LIN {X 0,Y 154.396,Z 231.863,A -85,B 0,C 180,E1 -25600.747,E2 -25600.747} C_VEL
LIN {X 0,Y 155.915,Z 236.605,A -85,B 0,C 180,E1 -25601.641,E2 -25601.641} C_VEL
LIN {X 0,Y 156.378,Z 245.915,A -85,B 0,C 180,E1 -25602.409,E2 -25602.409} C_VEL
LIN {X 0,Y 153.594,Z 283.863,A -85,B 0,C 180,E1 -25603.923,E2 -25603.923} C_VEL
LIN {X 0,Y 151.68,Z 296.984,A -85,B 0,C 180,E1 -25604.847,E2 -25604.847} C_VEL
LIN {X 0,Y 149.016,Z 309.429,A -85,B 0,C 180,E1 -25606.16,E2 -25606.16} C_VEL
LIN {X 0,Y 145.588,Z 321.476,A -85,B 0,C 180,E1 -25607.953,E2 -25607.953} C_VEL
LIN {X 0,Y 141.539,Z 332.987,A -85,B 0,C 180,E1 -25610.265,E2 -25610.265} C_VEL
LIN {X 0,Y 137.43,Z 343.378,A -85,B 0,C 180,E1 -25613.071,E2 -25613.071} C_VEL
LIN {X 0,Y 133.22,Z 352.693,A -85,B 0,C 180,E1 -25616.367,E2 -25616.367} C_VEL
LIN {X 0,Y 128.946,Z 361.751,A -85,B 0,C 180,E1 -25620.628,E2 -25620.628} C_VEL
LIN {X 0,Y 126.065,Z 367.927,A -85,B 0,C 180,E1 -25624.406,E2 -25624.406} C_VEL
LIN {X 0,Y 122.722,Z 374.878,A -85,B 0,C 180,E1 -25629.907,E2 -25629.907} C_VEL
LIN {X 0,Y 120.764,Z 379.462,A -85,B 0,C 180,E1 -25634.822,E2 -25634.822} C_VEL
LIN {X 0,Y 119.733,Z 382.952,A -85,B 0,C 180,E1 -25639.861,E2 -25639.861} C_VEL
LIN {X 0,Y 119.445,Z 384.69,A -85,B 0,C 180,E1 -25643.245,E2 -25643.245} C_VEL
LIN {X 0,Y 119.517,Z 386.571,A -85,B 0,C 180,E1 -25648.487,E2 -25648.487} C_VEL
LIN {X 0,Y 119.507,Z 387.154,A -85,B 0,C 180,E1 -25651.307,E2 -25651.307} C_VEL
LIN {X 0,Y 119.405,Z 387.457,A -85,B 0,C 180,E1 -25656.763,E2 -25656.763} C_VEL
LIN {X 0,Y 120.43,Z 386.4,A -85,B 0,C 180,E1 -25663.502,E2 -25663.502} C_VEL
LIN {X 0,Y 121.441,Z 385.287,A -85,B 0,C 180,E1 -25666.822,E2 -25666.822} C_VEL
LIN {X 0,Y 122.892,Z 383.731,A -85,B 0,C 180,E1 -25670.071,E2 -25670.071} C_VEL
LIN {X 0,Y 125.89,Z 380.63,A -85,B 0,C 180,E1 -25674.755,E2 -25674.755} C_VEL
LIN {X 0,Y 129.628,Z 376.486,A -85,B 0,C 180,E1 -25679.209,E2 -25679.209} C_VEL
LIN {X 0,Y 132.399,Z 373.117,A -85,B 0,C 180,E1 -25682.022,E2 -25682.022} C_VEL
LIN {X 0,Y 134.104,Z 370.343,A -85,B 0,C 180,E1 -25684.147,E2 -25684.147} C_VEL
LIN {X 0,Y 135.626,Z 365.454,A -85,B 0,C 180,E1 -25687.762,E2 -25687.762} C_VEL
LIN {X 0,Y 137.518,Z 359.972,A -85,B 0,C 180,E1 -25691.126,E2 -25691.126} C_VEL
LIN {X 0,Y 139.702,Z 356.26,A -85,B 0,C 180,E1 -25692.791,E2 -25692.791} C_VEL
LIN {X 0,Y 145.248,Z 347.956,A -85,B 0,C 180,E1 -25695.539,E2 -25695.539} C_VEL
LIN {X 0,Y 151.17,Z 337.757,A -85,B 0,C 180,E1 -25698.063,E2 -25698.063} C_VEL
LIN {X 0,Y 156.791,Z 326.24,A -85,B 0,C 180,E1 -25700.142,E2 -25700.142} C_VEL
LIN {X 0,Y 161.312,Z 314.911,A -85,B 0,C 180,E1 -25701.651,E2 -25701.651} C_VEL
LIN {X 0,Y 164.907,Z 303.329,A -85,B 0,C 180,E1 -25702.792,E2 -25702.792} C_VEL
LIN {X 0,Y 167.865,Z 289.908,A -85,B 0,C 180,E1 -25703.72,E2 -25703.72} C_VEL
LIN {X 0,Y 169.681,Z 276.62,A -85,B 0,C 180,E1 -25704.287,E2 -25704.287} C_VEL
LIN {X 0,Y 171.084,Z 259.051,A -85,B 0,C 180,E1 -25704.893,E2 -25704.893} C_VEL
LIN {X 0,Y 167.769,Z 249.581,A -85,B 0,C 180,E1 -25707.45,E2 -25707.45} C_VEL
LIN {X 0,Y 163.733,Z 239.799,A -85,B 0,C 180,E1 -25710.853,E2 -25710.853} C_VEL
LIN {X 0,Y 160.299,Z 232.342,A -85,B 0,C 180,E1 -25714.165,E2 -25714.165} C_VEL
LIN {X 0,Y 157.633,Z 227.099,A -85,B 0,C 180,E1 -25717.125,E2 -25717.125} C_VEL
LIN {X 0,Y 155.962,Z 224.434,A -85,B 0,C 180,E1 -25719.18,E2 -25719.18} C_VEL
LIN {X 0,Y 153.376,Z 220.422,A -85,B 0,C 180,E1 -25722.984,E2 -25722.984} C_VEL
LIN {X 0,Y 151.058,Z 217.466,A -85,B 0,C 180,E1 -25727.503,E2 -25727.503} C_VEL
LIN {X 0,Y 150.287,Z 215.488,A -85,B 0,C 180,E1 -25729.9,E2 -25729.9} C_VEL
LIN {X 0,Y 149.092,Z 214.312,A -85,B 0,C 180,E1 -25740,E2 -25740} C_VEL
LIN {X 0,Y 150.553,Z 215.702,A -85,B 0,C 180,E1 -25746.534,E2 -25746.534} C_VEL
LIN {X 0,Y 152.095,Z 219.04,A -85,B 0,C 180,E1 -25750.462,E2 -25750.462} C_VEL
LIN {X 0,Y 153.647,Z 220.772,A -85,B 0,C 180,E1 -25753.127,E2 -25753.127} C_VEL
LIN {X 0,Y 156.237,Z 224.739,A -85,B 0,C 180,E1 -25756.833,E2 -25756.833} C_VEL
LIN {X 0,Y 159.48,Z 229.84,A -85,B 0,C 180,E1 -25760.549,E2 -25760.549} C_VEL
LIN {X 0,Y 163.204,Z 235.852,A -85,B 0,C 180,E1 -25764.075,E2 -25764.075} C_VEL
LIN {X 0,Y 167.896,Z 244.453,A -85,B 0,C 180,E1 -25767.873,E2 -25767.873} C_VEL
LIN {X 0,Y 171.689,Z 252.135,A -85,B 0,C 180,E1 -25770.571,E2 -25770.571} C_VEL
LIN {X 0,Y 169.601,Z 275.061,A -85,B 0,C 180,E1 -25771.384,E2 -25771.384} C_VEL
LIN {X 0,Y 167.292,Z 288.542,A -85,B 0,C 180,E1 -25772.211,E2 -25772.211} C_VEL
LIN {X 0,Y 164.053,Z 301.073,A -85,B 0,C 180,E1 -25773.342,E2 -25773.342} C_VEL
LIN {X 0,Y 159.915,Z 313.018,A -85,B 0,C 180,E1 -25774.843,E2 -25774.843} C_VEL
LIN {X 0,Y 154.885,Z 324.813,A -85,B 0,C 180,E1 -25776.891,E2 -25776.891} C_VEL
LIN {X 0,Y 149.638,Z 334.818,A -85,B 0,C 180,E1 -25779.197,E2 -25779.197} C_VEL
LIN {X 0,Y 144.035,Z 343.862,A -85,B 0,C 180,E1 -25781.915,E2 -25781.915} C_VEL
LIN {X 0,Y 138.855,Z 351.308,A -85,B 0,C 180,E1 -25784.877,E2 -25784.877} C_VEL
LIN {X 0,Y 133.231,Z 358.599,A -85,B 0,C 180,E1 -25788.744,E2 -25788.744} C_VEL
LIN {X 0,Y 128.01,Z 364.422,A -85,B 0,C 180,E1 -25792.846,E2 -25792.846} C_VEL
LIN {X 0,Y 123.515,Z 368.987,A -85,B 0,C 180,E1 -25797.276,E2 -25797.276} C_VEL
LIN {X 0,Y 119.689,Z 372.445,A -85,B 0,C 180,E1 -25801.979,E2 -25801.979} C_VEL
LIN {X 0,Y 117.597,Z 374.173,A -85,B 0,C 180,E1 -25805.267,E2 -25805.267} C_VEL
LIN {X 0,Y 114.444,Z 376.385,A -85,B 0,C 180,E1 -25812.115,E2 -25812.115} C_VEL
LIN {X 0,Y 113.499,Z 376.9,A -85,B 0,C 180,E1 -25815.656,E2 -25815.656} C_VEL
LIN {X 0,Y 112.872,Z 376.986,A -85,B 0,C 180,E1 -25819.231,E2 -25819.231} C_VEL
LIN {X 0,Y 112.572,Z 376.683,A -85,B 0,C 180,E1 -25822.824,E2 -25822.824} C_VEL
LIN {X 0,Y 112.532,Z 375.642,A -85,B 0,C 180,E1 -25827.804,E2 -25827.804} C_VEL
LIN {X 0,Y 113.178,Z 373.447,A -85,B 0,C 180,E1 -25833.557,E2 -25833.557} C_VEL
LIN {X 0,Y 114.512,Z 370.428,A -85,B 0,C 180,E1 -25838.823,E2 -25838.823} C_VEL
LIN {X 0,Y 116.535,Z 366.376,A -85,B 0,C 180,E1 -25843.956,E2 -25843.956} C_VEL
LIN {X 0,Y 119.949,Z 360.16,A -85,B 0,C 180,E1 -25849.685,E2 -25849.685} C_VEL
LIN {X 0,Y 123.611,Z 353.4,A -85,B 0,C 180,E1 -25854.34,E2 -25854.34} C_VEL
LIN {X 0,Y 127.95,Z 344.971,A -85,B 0,C 180,E1 -25858.722,E2 -25858.722} C_VEL
LIN {X 0,Y 132.069,Z 336.303,A -85,B 0,C 180,E1 -25862.147,E2 -25862.147} C_VEL
LIN {X 0,Y 136.576,Z 325.633,A -85,B 0,C 180,E1 -25865.37,E2 -25865.37} C_VEL
LIN {X 0,Y 140.367,Z 314.989,A -85,B 0,C 180,E1 -25867.827,E2 -25867.827} C_VEL
LIN {X 0,Y 143.89,Z 303.05,A -85,B 0,C 180,E1 -25869.867,E2 -25869.867} C_VEL
LIN {X 0,Y 146.736,Z 290.607,A -85,B 0,C 180,E1 -25871.415,E2 -25871.415} C_VEL
LIN {X 0,Y 148.853,Z 277.413,A -85,B 0,C 180,E1 -25872.523,E2 -25872.523} C_VEL
LIN {X 0,Y 150.177,Z 262.193,A -85,B 0,C 180,E1 -25873.276,E2 -25873.276} C_VEL
LIN {X 0,Y 152.176,Z 234.348,A -85,B 0,C 180,E1 -25874.363,E2 -25874.363} C_VEL
LIN {X 0,Y 146.942,Z 223.579,A -85,B 0,C 180,E1 -25877.424,E2 -25877.424} C_VEL
LIN {X 0,Y 142.234,Z 215.384,A -85,B 0,C 180,E1 -25880.444,E2 -25880.444} C_VEL
LIN {X 0,Y 137.619,Z 208.218,A -85,B 0,C 180,E1 -25883.771,E2 -25883.771} C_VEL
LIN {X 0,Y 134.714,Z 204.022,A -85,B 0,C 180,E1 -25886.122,E2 -25886.122} C_VEL
LIN {X 0,Y 132.254,Z 200.514,A -85,B 0,C 180,E1 -25888.33,E2 -25888.33} C_VEL
LIN {X 0,Y 129.549,Z 196.833,A -85,B 0,C 180,E1 -25891.04,E2 -25891.04} C_VEL
LIN {X 0,Y 128.745,Z 195.852,A -85,B 0,C 180,E1 -25891.906,E2 -25891.906} C_VEL
LIN {X 0,Y 126.275,Z 193.061,A -85,B 0,C 180,E1 -25894.806,E2 -25894.806} C_VEL
LIN {X 0,Y 125.163,Z 190.919,A -85,B 0,C 180,E1 -25896.417,E2 -25896.417} C_VEL
LIN {X 0,Y 122.32,Z 188.789,A -85,B 0,C 180,E1 -25900.708,E2 -25900.708} C_VEL
LIN {X 0,Y 120.813,Z 185.857,A -85,B 0,C 180,E1 -25904.067,E2 -25904.067} C_VEL
LIN {X 0,Y 120.553,Z 185.187,A -85,B 0,C 180,E1 -25904.791,E2 -25904.791} C_VEL
LIN {X 0,Y 117.979,Z 183.461,A -85,B 0,C 180,E1 -25918.293,E2 -25918.293} C_VEL
LIN {X 0,Y 118.187,Z 183.542,A -85,B 0,C 180,E1 -25920.851,E2 -25920.851} C_VEL
LIN {X 0,Y 120.921,Z 185.41,A -85,B 0,C 180,E1 -25930.436,E2 -25930.436} C_VEL
LIN {X 0,Y 121.931,Z 188.11,A -85,B 0,C 180,E1 -25932.912,E2 -25932.912} C_VEL
LIN {X 0,Y 124.382,Z 190.53,A -85,B 0,C 180,E1 -25936.938,E2 -25936.938} C_VEL
LIN {X 0,Y 125.444,Z 191.294,A -85,B 0,C 180,E1 -25938.369,E2 -25938.369} C_VEL
LIN {X 0,Y 127.207,Z 194.369,A -85,B 0,C 180,E1 -25940.768,E2 -25940.768} C_VEL
LIN {X 0,Y 129.466,Z 196.653,A -85,B 0,C 180,E1 -25943.255,E2 -25943.255} C_VEL
LIN {X 0,Y 132.137,Z 200.357,A -85,B 0,C 180,E1 -25945.952,E2 -25945.952} C_VEL
LIN {X 0,Y 136.383,Z 206.271,A -85,B 0,C 180,E1 -25949.635,E2 -25949.635} C_VEL
LIN {X 0,Y 139.737,Z 211.368,A -85,B 0,C 180,E1 -25952.195,E2 -25952.195} C_VEL
LIN {X 0,Y 143.818,Z 219.923,A -85,B 0,C 180,E1 -25955.15,E2 -25955.15} C_VEL
LIN {X 0,Y 147.828,Z 229.624,A -85,B 0,C 180,E1 -25957.823,E2 -25957.823} C_VEL
LIN {X 0,Y 151.055,Z 238.927,A -85,B 0,C 180,E1 -25959.88,E2 -25959.88} C_VEL
LIN {X 0,Y 151.318,Z 247.608,A -85,B 0,C 180,E1 -25960.581,E2 -25960.581} C_VEL
LIN {X 0,Y 148.549,Z 283.444,A -85,B 0,C 180,E1 -25962.022,E2 -25962.022} C_VEL
LIN {X 0,Y 146.599,Z 296.41,A -85,B 0,C 180,E1 -25962.94,E2 -25962.94} C_VEL
LIN {X 0,Y 143.994,Z 308.361,A -85,B 0,C 180,E1 -25964.209,E2 -25964.209} C_VEL
LIN {X 0,Y 140.384,Z 320.627,A -85,B 0,C 180,E1 -25966.008,E2 -25966.008} C_VEL
LIN {X 0,Y 136.133,Z 332.233,A -85,B 0,C 180,E1 -25968.346,E2 -25968.346} C_VEL
LIN {X 0,Y 131.799,Z 342.7,A -85,B 0,C 180,E1 -25971.208,E2 -25971.208} C_VEL
LIN {X 0,Y 127.328,Z 352.097,A -85,B 0,C 180,E1 -25974.585,E2 -25974.585} C_VEL
LIN {X 0,Y 122.771,Z 361.201,A -85,B 0,C 180,E1 -25978.993,E2 -25978.993} C_VEL
LIN {X 0,Y 119.049,Z 368.542,A -85,B 0,C 180,E1 -25983.724,E2 -25983.724} C_VEL
LIN {X 0,Y 116.032,Z 374.411,A -85,B 0,C 180,E1 -25988.694,E2 -25988.694} C_VEL
LIN {X 0,Y 113.887,Z 379.029,A -85,B 0,C 180,E1 -25993.881,E2 -25993.881} C_VEL
LIN {X 0,Y 112.724,Z 382.546,A -85,B 0,C 180,E1 -25999.223,E2 -25999.223} C_VEL
LIN {X 0,Y 112.361,Z 384.304,A -85,B 0,C 180,E1 -26002.817,E2 -26002.817} C_VEL
LIN {X 0,Y 112.459,Z 386.396,A -85,B 0,C 180,E1 -26009.198,E2 -26009.198} C_VEL
LIN {X 0,Y 112.333,Z 387.077,A -85,B 0,C 180,E1 -26013.59,E2 -26013.59} C_VEL
LIN {X 0,Y 112.722,Z 386.814,A -85,B 0,C 180,E1 -26020.784,E2 -26020.784} C_VEL
LIN {X 0,Y 114.619,Z 385.013,A -85,B 0,C 180,E1 -26027.856,E2 -26027.856} C_VEL
LIN {X 0,Y 116.233,Z 383.48,A -85,B 0,C 180,E1 -26031.275,E2 -26031.275} C_VEL
LIN {X 0,Y 119.435,Z 380.407,A -85,B 0,C 180,E1 -26036.192,E2 -26036.192} C_VEL
LIN {X 0,Y 123.44,Z 376.294,A -85,B 0,C 180,E1 -26040.828,E2 -26040.828} C_VEL
LIN {X 0,Y 128.908,Z 370.011,A -85,B 0,C 180,E1 -26045.883,E2 -26045.883} C_VEL
LIN {X 0,Y 134.522,Z 363.203,A -85,B 0,C 180,E1 -26049.794,E2 -26049.794} C_VEL
LIN {X 0,Y 139.702,Z 356.26,A -85,B 0,C 180,E1 -26052.791,E2 -26052.791} C_VEL
LIN {X 0,Y 141.936,Z 352.367,A -85,B 0,C 180,E1 -26054.355,E2 -26054.355} C_VEL
LIN {X 0,Y 144.244,Z 345.749,A -85,B 0,C 180,E1 -26057.168,E2 -26057.168} C_VEL
LIN {X 0,Y 146.516,Z 338.649,A -85,B 0,C 180,E1 -26059.74,E2 -26059.74} C_VEL
LIN {X 0,Y 148.598,Z 333.995,A -85,B 0,C 180,E1 -26060.895,E2 -26060.895} C_VEL
LIN {X 0,Y 153.67,Z 323.487,A -85,B 0,C 180,E1 -26062.624,E2 -26062.624} C_VEL
LIN {X 0,Y 158.3,Z 311.363,A -85,B 0,C 180,E1 -26064.122,E2 -26064.122} C_VEL
LIN {X 0,Y 162.082,Z 298.685,A -85,B 0,C 180,E1 -26065.202,E2 -26065.202} C_VEL
LIN {X 0,Y 164.705,Z 285.496,A -85,B 0,C 180,E1 -26065.988,E2 -26065.988} C_VEL
LIN {X 0,Y 166.668,Z 267.36,A -85,B 0,C 180,E1 -26066.623,E2 -26066.623} C_VEL
LIN {X 0,Y 167.099,Z 261.511,A -85,B 0,C 180,E1 -26066.855,E2 -26066.855} C_VEL
LIN {X 0,Y 163.705,Z 251.8,A -85,B 0,C 180,E1 -26069.758,E2 -26069.758} C_VEL
LIN {X 0,Y 160.092,Z 242.761,A -85,B 0,C 180,E1 -26073.213,E2 -26073.213} C_VEL
LIN {X 0,Y 157.735,Z 237.548,A -85,B 0,C 180,E1 -26075.755,E2 -26075.755} C_VEL
LIN {X 0,Y 155.773,Z 233.325,A -85,B 0,C 180,E1 -26078.159,E2 -26078.159} C_VEL
LIN {X 0,Y 154.088,Z 230.59,A -85,B 0,C 180,E1 -26080.397,E2 -26080.397} C_VEL
LIN {X 0,Y 151.914,Z 227.078,A -85,B 0,C 180,E1 -26083.885,E2 -26083.885} C_VEL
LIN {X 0,Y 149.793,Z 223.969,A -85,B 0,C 180,E1 -26088.498,E2 -26088.498} C_VEL
LIN {X 0,Y 149.319,Z 222.497,A -85,B 0,C 180,E1 -26090.176,E2 -26090.176} C_VEL
LIN {X 0,Y 148.222,Z 221.381,A -85,B 0,C 180,E1 -26100,E2 -26100} C_VEL
LIN {X 0,Y 149.503,Z 222.698,A -85,B 0,C 180,E1 -26106.072,E2 -26106.072} C_VEL
LIN {X 0,Y 150.944,Z 225.915,A -85,B 0,C 180,E1 -26109.971,E2 -26109.971} C_VEL
LIN {X 0,Y 152.366,Z 227.715,A -85,B 0,C 180,E1 -26112.572,E2 -26112.572} C_VEL
LIN {X 0,Y 155.324,Z 232.491,A -85,B 0,C 180,E1 -26116.935,E2 -26116.935} C_VEL
LIN {X 0,Y 157.845,Z 236.636,A -85,B 0,C 180,E1 -26119.91,E2 -26119.91} C_VEL
LIN {X 0,Y 161.138,Z 242.306,A -85,B 0,C 180,E1 -26123.212,E2 -26123.212} C_VEL
LIN {X 0,Y 165.005,Z 249.718,A -85,B 0,C 180,E1 -26126.565,E2 -26126.565} C_VEL
LIN {X 0,Y 167.661,Z 255.284,A -85,B 0,C 180,E1 -26128.632,E2 -26128.632} C_VEL
LIN {X 0,Y 165.761,Z 275.351,A -85,B 0,C 180,E1 -26129.357,E2 -26129.357} C_VEL
LIN {X 0,Y 163.405,Z 288.528,A -85,B 0,C 180,E1 -26130.136,E2 -26130.136} C_VEL
LIN {X 0,Y 160.245,Z 300.653,A -85,B 0,C 180,E1 -26131.212,E2 -26131.212} C_VEL
LIN {X 0,Y 156.006,Z 312.631,A -85,B 0,C 180,E1 -26132.674,E2 -26132.674} C_VEL
LIN {X 0,Y 150.712,Z 324.669,A -85,B 0,C 180,E1 -26134.723,E2 -26134.723} C_VEL
LIN {X 0,Y 145.225,Z 334.786,A -85,B 0,C 180,E1 -26137.01,E2 -26137.01} C_VEL
LIN {X 0,Y 139.362,Z 343.89,A -85,B 0,C 180,E1 -26139.728,E2 -26139.728} C_VEL
LIN {X 0,Y 133.04,Z 352.479,A -85,B 0,C 180,E1 -26143.202,E2 -26143.202} C_VEL
LIN {X 0,Y 126.978,Z 359.811,A -85,B 0,C 180,E1 -26147.308,E2 -26147.308} C_VEL
LIN {X 0,Y 120.689,Z 366.229,A -85,B 0,C 180,E1 -26152.303,E2 -26152.303} C_VEL
LIN {X 0,Y 116.082,Z 370.446,A -85,B 0,C 180,E1 -26156.979,E2 -26156.979} C_VEL
LIN {X 0,Y 113.404,Z 372.675,A -85,B 0,C 180,E1 -26160.275,E2 -26160.275} C_VEL
LIN {X 0,Y 111.122,Z 374.433,A -85,B 0,C 180,E1 -26163.719,E2 -26163.719} C_VEL
LIN {X 0,Y 107.653,Z 376.674,A -85,B 0,C 180,E1 -26170.945,E2 -26170.945} C_VEL
LIN {X 0,Y 106.57,Z 377.209,A -85,B 0,C 180,E1 -26174.702,E2 -26174.702} C_VEL
LIN {X 0,Y 105.858,Z 377.319,A -85,B 0,C 180,E1 -26178.508,E2 -26178.508} C_VEL
LIN {X 0,Y 105.503,Z 377.03,A -85,B 0,C 180,E1 -26182.34,E2 -26182.34} C_VEL
LIN {X 0,Y 105.466,Z 375.819,A -85,B 0,C 180,E1 -26188.325,E2 -26188.325} C_VEL
LIN {X 0,Y 106.095,Z 373.852,A -85,B 0,C 180,E1 -26193.795,E2 -26193.795} C_VEL
LIN {X 0,Y 107.522,Z 370.864,A -85,B 0,C 180,E1 -26199.401,E2 -26199.401} C_VEL
LIN {X 0,Y 109.681,Z 366.845,A -85,B 0,C 180,E1 -26204.847,E2 -26204.847} C_VEL
LIN {X 0,Y 113.311,Z 360.665,A -85,B 0,C 180,E1 -26210.89,E2 -26210.89} C_VEL
LIN {X 0,Y 117.215,Z 353.945,A -85,B 0,C 180,E1 -26215.762,E2 -26215.762} C_VEL
LIN {X 0,Y 121.806,Z 345.588,A -85,B 0,C 180,E1 -26220.318,E2 -26220.318} C_VEL
LIN {X 0,Y 126.159,Z 336.977,A -85,B 0,C 180,E1 -26223.85,E2 -26223.85} C_VEL
LIN {X 0,Y 130.894,Z 326.378,A -85,B 0,C 180,E1 -26227.155,E2 -26227.155} C_VEL
LIN {X 0,Y 134.866,Z 315.848,A -85,B 0,C 180,E1 -26229.665,E2 -26229.665} C_VEL
LIN {X 0,Y 138.557,Z 304.09,A -85,B 0,C 180,E1 -26231.734,E2 -26231.734} C_VEL
LIN {X 0,Y 141.533,Z 291.87,A -85,B 0,C 180,E1 -26233.3,E2 -26233.3} C_VEL
LIN {X 0,Y 143.847,Z 278.493,A -85,B 0,C 180,E1 -26234.474,E2 -26234.474} C_VEL
LIN {X 0,Y 145.295,Z 263.241,A -85,B 0,C 180,E1 -26235.245,E2 -26235.245} C_VEL
LIN {X 0,Y 147.22,Z 236.744,A -85,B 0,C 180,E1 -26236.32,E2 -26236.32} C_VEL
LIN {X 0,Y 142.32,Z 226.723,A -85,B 0,C 180,E1 -26239.469,E2 -26239.469} C_VEL
LIN {X 0,Y 138.007,Z 219.078,A -85,B 0,C 180,E1 -26242.539,E2 -26242.539} C_VEL
LIN {X 0,Y 134.281,Z 213.216,A -85,B 0,C 180,E1 -26245.499,E2 -26245.499} C_VEL
LIN {X 0,Y 131.743,Z 209.345,A -85,B 0,C 180,E1 -26247.76,E2 -26247.76} C_VEL
LIN {X 0,Y 129.879,Z 206.631,A -85,B 0,C 180,E1 -26249.573,E2 -26249.573} C_VEL
LIN {X 0,Y 126.805,Z 202.306,A -85,B 0,C 180,E1 -26252.946,E2 -26252.946} C_VEL
LIN {X 0,Y 124.438,Z 199.456,A -85,B 0,C 180,E1 -26255.939,E2 -26255.939} C_VEL
LIN {X 0,Y 123.218,Z 197.487,A -85,B 0,C 180,E1 -26257.789,E2 -26257.789} C_VEL
LIN {X 0,Y 120.731,Z 195.214,A -85,B 0,C 180,E1 -26261.985,E2 -26261.985} C_VEL
LIN {X 0,Y 119.358,Z 192.153,A -85,B 0,C 180,E1 -26265.507,E2 -26265.507} C_VEL
LIN {X 0,Y 117.085,Z 190.624,A -85,B 0,C 180,E1 -26276.558,E2 -26276.558} C_VEL
LIN {X 0,Y 117.275,Z 190.529,A -85,B 0,C 180,E1 -26280.429,E2 -26280.429} C_VEL
LIN {X 0,Y 119.573,Z 192.251,A -85,B 0,C 180,E1 -26289.408,E2 -26289.408} C_VEL
LIN {X 0,Y 120.835,Z 195.247,A -85,B 0,C 180,E1 -26292.598,E2 -26292.598} C_VEL
LIN {X 0,Y 123.728,Z 198.002,A -85,B 0,C 180,E1 -26297.35,E2 -26297.35} C_VEL
LIN {X 0,Y 125.768,Z 201.304,A -85,B 0,C 180,E1 -26300.228,E2 -26300.228} C_VEL
LIN {X 0,Y 127.435,Z 203.105,A -85,B 0,C 180,E1 -26302.174,E2 -26302.174} C_VEL
LIN {X 0,Y 130.907,Z 208.098,A -85,B 0,C 180,E1 -26305.835,E2 -26305.835} C_VEL
LIN {X 0,Y 133.994,Z 212.655,A -85,B 0,C 180,E1 -26308.636,E2 -26308.636} C_VEL
LIN {X 0,Y 136.711,Z 216.991,A -85,B 0,C 180,E1 -26310.862,E2 -26310.862} C_VEL
LIN {X 0,Y 140.515,Z 225.459,A -85,B 0,C 180,E1 -26313.849,E2 -26313.849} C_VEL
LIN {X 0,Y 144.6,Z 235.956,A -85,B 0,C 180,E1 -26316.79,E2 -26316.79} C_VEL
LIN {X 0,Y 146.355,Z 241.629,A -85,B 0,C 180,E1 -26318.037,E2 -26318.037} C_VEL
LIN {X 0,Y 146.477,Z 248.428,A -85,B 0,C 180,E1 -26318.59,E2 -26318.59} C_VEL
LIN {X 0,Y 143.653,Z 283.313,A -85,B 0,C 180,E1 -26320.013,E2 -26320.013} C_VEL
LIN {X 0,Y 141.588,Z 296.322,A -85,B 0,C 180,E1 -26320.938,E2 -26320.938} C_VEL
LIN {X 0,Y 138.829,Z 308.413,A -85,B 0,C 180,E1 -26322.242,E2 -26322.242} C_VEL
LIN {X 0,Y 135.362,Z 319.771,A -85,B 0,C 180,E1 -26323.918,E2 -26323.918} C_VEL
LIN {X 0,Y 130.904,Z 331.476,A -85,B 0,C 180,E1 -26326.277,E2 -26326.277} C_VEL
LIN {X 0,Y 126.313,Z 342.016,A -85,B 0,C 180,E1 -26329.178,E2 -26329.178} C_VEL
LIN {X 0,Y 121.585,Z 351.498,A -85,B 0,C 180,E1 -26332.637,E2 -26332.637} C_VEL
LIN {X 0,Y 116.703,Z 360.648,A -85,B 0,C 180,E1 -26337.185,E2 -26337.185} C_VEL
LIN {X 0,Y 112.715,Z 368.033,A -85,B 0,C 180,E1 -26342.123,E2 -26342.123} C_VEL
LIN {X 0,Y 109.407,Z 373.939,A -85,B 0,C 180,E1 -26347.334,E2 -26347.334} C_VEL
LIN {X 0,Y 107.026,Z 378.59,A -85,B 0,C 180,E1 -26352.817,E2 -26352.817} C_VEL
LIN {X 0,Y 105.736,Z 382.137,A -85,B 0,C 180,E1 -26358.502,E2 -26358.502} C_VEL
LIN {X 0,Y 105.291,Z 383.919,A -85,B 0,C 180,E1 -26362.332,E2 -26362.332} C_VEL
LIN {X 0,Y 105.243,Z 385.272,A -85,B 0,C 180,E1 -26366.175,E2 -26366.175} C_VEL
LIN {X 0,Y 105.42,Z 386.22,A -85,B 0,C 180,E1 -26370.004,E2 -26370.004} C_VEL
LIN {X 0,Y 105.239,Z 386.739,A -85,B 0,C 180,E1 -26373.833,E2 -26373.833} C_VEL
LIN {X 0,Y 105.742,Z 386.509,A -85,B 0,C 180,E1 -26381.505,E2 -26381.505} C_VEL
LIN {X 0,Y 107.843,Z 384.736,A -85,B 0,C 180,E1 -26389.02,E2 -26389.02} C_VEL
LIN {X 0,Y 109.636,Z 383.23,A -85,B 0,C 180,E1 -26392.623,E2 -26392.623} C_VEL
LIN {X 0,Y 113.07,Z 380.185,A -85,B 0,C 180,E1 -26397.789,E2 -26397.789} C_VEL
LIN {X 0,Y 117.342,Z 376.101,A -85,B 0,C 180,E1 -26402.621,E2 -26402.621} C_VEL
LIN {X 0,Y 123.207,Z 369.854,A -85,B 0,C 180,E1 -26407.825,E2 -26407.825} C_VEL
LIN {X 0,Y 129.131,Z 363.084,A -85,B 0,C 180,E1 -26411.817,E2 -26411.817} C_VEL
LIN {X 0,Y 135.706,Z 354.701,A -85,B 0,C 180,E1 -26415.408,E2 -26415.408} C_VEL
LIN {X 0,Y 141.54,Z 346.081,A -85,B 0,C 180,E1 -26418.146,E2 -26418.146} C_VEL
LIN {X 0,Y 147.798,Z 335.478,A -85,B 0,C 180,E1 -26420.601,E2 -26420.601} C_VEL
LIN {X 0,Y 148.598,Z 333.995,A -85,B 0,C 180,E1 -26420.895,E2 -26420.895} C_VEL
LIN {X 0,Y 150.631,Z 329.187,A -85,B 0,C 180,E1 -26421.965,E2 -26421.965} C_VEL
LIN {X 0,Y 152.667,Z 321.174,A -85,B 0,C 180,E1 -26424.043,E2 -26424.043} C_VEL
LIN {X 0,Y 154.37,Z 312.79,A -85,B 0,C 180,E1 -26425.907,E2 -26425.907} C_VEL
LIN {X 0,Y 155.798,Z 307.406,A -85,B 0,C 180,E1 -26426.628,E2 -26426.628} C_VEL
LIN {X 0,Y 159.435,Z 293.765,A -85,B 0,C 180,E1 -26427.693,E2 -26427.693} C_VEL
LIN {X 0,Y 161.714,Z 281.24,A -85,B 0,C 180,E1 -26428.293,E2 -26428.293} C_VEL
LIN {X 0,Y 163.3,Z 264.164,A -85,B 0,C 180,E1 -26428.906,E2 -26428.906} C_VEL
LIN {X 0,Y 160.421,Z 255.632,A -85,B 0,C 180,E1 -26431.652,E2 -26431.652} C_VEL
LIN {X 0,Y 157.551,Z 247.953,A -85,B 0,C 180,E1 -26434.71,E2 -26434.71} C_VEL
LIN {X 0,Y 154.769,Z 241.392,A -85,B 0,C 180,E1 -26438.108,E2 -26438.108} C_VEL
LIN {X 0,Y 153.092,Z 237.896,A -85,B 0,C 180,E1 -26440.463,E2 -26440.463} C_VEL
LIN {X 0,Y 150.507,Z 233.754,A -85,B 0,C 180,E1 -26444.772,E2 -26444.772} C_VEL
LIN {X 0,Y 148.533,Z 230.359,A -85,B 0,C 180,E1 -26449.655,E2 -26449.655} C_VEL
LIN {X 0,Y 148.297,Z 229.504,A -85,B 0,C 180,E1 -26450.628,E2 -26450.628} C_VEL
LIN {X 0,Y 147.242,Z 228.554,A -85,B 0,C 180,E1 -26457.264,E2 -26457.264} C_VEL
LIN {X 0,Y 147.412,Z 228.599,A -85,B 0,C 180,E1 -26460.683,E2 -26460.683} C_VEL
LIN {X 0,Y 148.456,Z 229.752,A -85,B 0,C 180,E1 -26465.604,E2 -26465.604} C_VEL
LIN {X 0,Y 150.066,Z 233.174,A -85,B 0,C 180,E1 -26470.03,E2 -26470.03} C_VEL
LIN {X 0,Y 151.054,Z 234.527,A -85,B 0,C 180,E1 -26471.915,E2 -26471.915} C_VEL
LIN {X 0,Y 153.596,Z 238.809,A -85,B 0,C 180,E1 -26475.935,E2 -26475.935} C_VEL
LIN {X 0,Y 156.121,Z 243.251,A -85,B 0,C 180,E1 -26479.134,E2 -26479.134} C_VEL
LIN {X 0,Y 159.479,Z 249.482,A -85,B 0,C 180,E1 -26482.692,E2 -26482.692} C_VEL
LIN {X 0,Y 162.988,Z 256.652,A -85,B 0,C 180,E1 -26485.89,E2 -26485.89} C_VEL
LIN {X 0,Y 163.828,Z 258.556,A -85,B 0,C 180,E1 -26486.605,E2 -26486.605} C_VEL
LIN {X 0,Y 162.024,Z 276.337,A -85,B 0,C 180,E1 -26487.261,E2 -26487.261} C_VEL
LIN {X 0,Y 159.544,Z 289.564,A -85,B 0,C 180,E1 -26488.055,E2 -26488.055} C_VEL
LIN {X 0,Y 155.975,Z 302.264,A -85,B 0,C 180,E1 -26489.187,E2 -26489.187} C_VEL
LIN {X 0,Y 151.416,Z 314.413,A -85,B 0,C 180,E1 -26490.702,E2 -26490.702} C_VEL
LIN {X 0,Y 146.112,Z 325.798,A -85,B 0,C 180,E1 -26492.671,E2 -26492.671} C_VEL
LIN {X 0,Y 141.034,Z 334.751,A -85,B 0,C 180,E1 -26494.689,E2 -26494.689} C_VEL
LIN {X 0,Y 134.905,Z 343.918,A -85,B 0,C 180,E1 -26497.392,E2 -26497.392} C_VEL
LIN {X 0,Y 129.14,Z 351.464,A -85,B 0,C 180,E1 -26500.364,E2 -26500.364} C_VEL
LIN {X 0,Y 122.799,Z 358.843,A -85,B 0,C 180,E1 -26504.321,E2 -26504.321} C_VEL
LIN {X 0,Y 116.907,Z 364.744,A -85,B 0,C 180,E1 -26508.599,E2 -26508.599} C_VEL
LIN {X 0,Y 111.707,Z 369.382,A -85,B 0,C 180,E1 -26513.292,E2 -26513.292} C_VEL
LIN {X 0,Y 107.062,Z 373.03,A -85,B 0,C 180,E1 -26518.582,E2 -26518.582} C_VEL
LIN {X 0,Y 104.739,Z 374.694,A -85,B 0,C 180,E1 -26521.982,E2 -26521.982} C_VEL
LIN {X 0,Y 100.913,Z 376.964,A -85,B 0,C 180,E1 -26529.618,E2 -26529.618} C_VEL
LIN {X 0,Y 99.681,Z 377.514,A -85,B 0,C 180,E1 -26533.616,E2 -26533.616} C_VEL
LIN {X 0,Y 98.876,Z 377.652,A -85,B 0,C 180,E1 -26537.684,E2 -26537.684} C_VEL
LIN {X 0,Y 98.444,Z 377.377,A -85,B 0,C 180,E1 -26541.788,E2 -26541.788} C_VEL
LIN {X 0,Y 98.406,Z 375.954,A -85,B 0,C 180,E1 -26549.076,E2 -26549.076} C_VEL
LIN {X 0,Y 99.017,Z 374.256,A -85,B 0,C 180,E1 -26554.066,E2 -26554.066} C_VEL
LIN {X 0,Y 100.547,Z 371.297,A -85,B 0,C 180,E1 -26560.06,E2 -26560.06} C_VEL
LIN {X 0,Y 102.858,Z 367.311,A -85,B 0,C 180,E1 -26565.857,E2 -26565.857} C_VEL
LIN {X 0,Y 106.734,Z 361.17,A -85,B 0,C 180,E1 -26572.244,E2 -26572.244} C_VEL
LIN {X 0,Y 110.888,Z 354.49,A -85,B 0,C 180,E1 -26577.351,E2 -26577.351} C_VEL
LIN {X 0,Y 115.763,Z 346.199,A -85,B 0,C 180,E1 -26582.083,E2 -26582.083} C_VEL
LIN {X 0,Y 120.353,Z 337.653,A -85,B 0,C 180,E1 -26585.724,E2 -26585.724} C_VEL
LIN {X 0,Y 125.353,Z 327.124,A -85,B 0,C 180,E1 -26589.1,E2 -26589.1} C_VEL
LIN {X 0,Y 129.516,Z 316.687,A -85,B 0,C 180,E1 -26591.657,E2 -26591.657} C_VEL
LIN {X 0,Y 133.38,Z 305.131,A -85,B 0,C 180,E1 -26593.75,E2 -26593.75} C_VEL
LIN {X 0,Y 136.506,Z 293.13,A -85,B 0,C 180,E1 -26595.323,E2 -26595.323} C_VEL
LIN {X 0,Y 138.922,Z 280.138,A -85,B 0,C 180,E1 -26596.51,E2 -26596.51} C_VEL
LIN {X 0,Y 140.348,Z 267.315,A -85,B 0,C 180,E1 -26597.233,E2 -26597.233} C_VEL
LIN {X 0,Y 142.527,Z 239.536,A -85,B 0,C 180,E1 -26598.338,E2 -26598.338} C_VEL
LIN {X 0,Y 138.274,Z 230.675,A -85,B 0,C 180,E1 -26601.355,E2 -26601.355} C_VEL
LIN {X 0,Y 134.301,Z 223.397,A -85,B 0,C 180,E1 -26604.482,E2 -26604.482} C_VEL
LIN {X 0,Y 129.875,Z 216.192,A -85,B 0,C 180,E1 -26608.475,E2 -26608.475} C_VEL
LIN {X 0,Y 127.443,Z 212.585,A -85,B 0,C 180,E1 -26610.994,E2 -26610.994} C_VEL
LIN {X 0,Y 124.925,Z 208.793,A -85,B 0,C 180,E1 -26613.993,E2 -26613.993} C_VEL
LIN {X 0,Y 122.478,Z 205.532,A -85,B 0,C 180,E1 -26617.383,E2 -26617.383} C_VEL
LIN {X 0,Y 121.747,Z 204.266,A -85,B 0,C 180,E1 -26618.592,E2 -26618.592} C_VEL
LIN {X 0,Y 119.328,Z 201.834,A -85,B 0,C 180,E1 -26623.011,E2 -26623.011} C_VEL
LIN {X 0,Y 118.174,Z 199.18,A -85,B 0,C 180,E1 -26626.238,E2 -26626.238} C_VEL
LIN {X 0,Y 116.218,Z 197.68,A -85,B 0,C 180,E1 -26636.533,E2 -26636.533} C_VEL
LIN {X 0,Y 116.444,Z 197.703,A -85,B 0,C 180,E1 -26640.864,E2 -26640.864} C_VEL
LIN {X 0,Y 118.356,Z 199.308,A -85,B 0,C 180,E1 -26648.644,E2 -26648.644} C_VEL
LIN {X 0,Y 119.752,Z 202.344,A -85,B 0,C 180,E1 -26652.283,E2 -26652.283} C_VEL
LIN {X 0,Y 122.121,Z 204.742,A -85,B 0,C 180,E1 -26656.4,E2 -26656.4} C_VEL
LIN {X 0,Y 124.296,Z 208.165,A -85,B 0,C 180,E1 -26659.616,E2 -26659.616} C_VEL
LIN {X 0,Y 125.586,Z 209.738,A -85,B 0,C 180,E1 -26661.223,E2 -26661.223} C_VEL
LIN {X 0,Y 128.597,Z 214.258,A -85,B 0,C 180,E1 -26664.627,E2 -26664.627} C_VEL
LIN {X 0,Y 131.672,Z 219.03,A -85,B 0,C 180,E1 -26667.618,E2 -26667.618} C_VEL
LIN {X 0,Y 133.73,Z 222.545,A -85,B 0,C 180,E1 -26669.442,E2 -26669.442} C_VEL
LIN {X 0,Y 137.463,Z 231.436,A -85,B 0,C 180,E1 -26672.631,E2 -26672.631} C_VEL
LIN {X 0,Y 140.931,Z 241.095,A -85,B 0,C 180,E1 -26675.362,E2 -26675.362} C_VEL
LIN {X 0,Y 141.807,Z 244.117,A -85,B 0,C 180,E1 -26676.052,E2 -26676.052} C_VEL
LIN {X 0,Y 141.806,Z 249.704,A -85,B 0,C 180,E1 -26676.493,E2 -26676.493} C_VEL
LIN {X 0,Y 138.998,Z 282.72,A -85,B 0,C 180,E1 -26677.833,E2 -26677.833} C_VEL
LIN {X 0,Y 136.796,Z 296.115,A -85,B 0,C 180,E1 -26678.786,E2 -26678.786} C_VEL
LIN {X 0,Y 133.841,Z 308.464,A -85,B 0,C 180,E1 -26680.127,E2 -26680.127} C_VEL
LIN {X 0,Y 129.929,Z 320.508,A -85,B 0,C 180,E1 -26681.953,E2 -26681.953} C_VEL
LIN {X 0,Y 125.293,Z 332.018,A -85,B 0,C 180,E1 -26684.347,E2 -26684.347} C_VEL
LIN {X 0,Y 120.475,Z 342.405,A -85,B 0,C 180,E1 -26687.306,E2 -26687.306} C_VEL
LIN {X 0,Y 115.988,Z 350.889,A -85,B 0,C 180,E1 -26690.494,E2 -26690.494} C_VEL
LIN {X 0,Y 110.775,Z 360.096,A -85,B 0,C 180,E1 -26695.185,E2 -26695.185} C_VEL
LIN {X 0,Y 107.751,Z 365.244,A -85,B 0,C 180,E1 -26698.552,E2 -26698.552} C_VEL
LIN {X 0,Y 103.949,Z 371.629,A -85,B 0,C 180,E1 -26703.934,E2 -26703.934} C_VEL
LIN {X 0,Y 100.945,Z 376.7,A -85,B 0,C 180,E1 -26709.632,E2 -26709.632} C_VEL
LIN {X 0,Y 99.107,Z 380.638,A -85,B 0,C 180,E1 -26715.633,E2 -26715.633} C_VEL
LIN {X 0,Y 98.249,Z 383.534,A -85,B 0,C 180,E1 -26721.779,E2 -26721.779} C_VEL
LIN {X 0,Y 98.134,Z 384.9,A -85,B 0,C 180,E1 -26725.897,E2 -26725.897} C_VEL
LIN {X 0,Y 98.314,Z 385.862,A -85,B 0,C 180,E1 -26730.004,E2 -26730.004} C_VEL
LIN {X 0,Y 98.133,Z 386.396,A -85,B 0,C 180,E1 -26734.111,E2 -26734.111} C_VEL
LIN {X 0,Y 98.232,Z 386.503,A -85,B 0,C 180,E1 -26738.23,E2 -26738.23} C_VEL
LIN {X 0,Y 99.712,Z 385.522,A -85,B 0,C 180,E1 -26746.379,E2 -26746.379} C_VEL
LIN {X 0,Y 101.121,Z 384.457,A -85,B 0,C 180,E1 -26750.338,E2 -26750.338} C_VEL
LIN {X 0,Y 103.11,Z 382.98,A -85,B 0,C 180,E1 -26754.143,E2 -26754.143} C_VEL
LIN {X 0,Y 106.812,Z 379.96,A -85,B 0,C 180,E1 -26759.573,E2 -26759.573} C_VEL
LIN {X 0,Y 111.396,Z 375.905,A -85,B 0,C 180,E1 -26764.601,E2 -26764.601} C_VEL
LIN {X 0,Y 117.661,Z 369.698,A -85,B 0,C 180,E1 -26769.953,E2 -26769.953} C_VEL
LIN {X 0,Y 123.907,Z 362.965,A -85,B 0,C 180,E1 -26774.016,E2 -26774.016} C_VEL
LIN {X 0,Y 130.82,Z 354.634,A -85,B 0,C 180,E1 -26777.623,E2 -26777.623} C_VEL
LIN {X 0,Y 136.91,Z 346.083,A -85,B 0,C 180,E1 -26780.357,E2 -26780.357} C_VEL
LIN {X 0,Y 143.41,Z 335.546,A -85,B 0,C 180,E1 -26782.786,E2 -26782.786} C_VEL
LIN {X 0,Y 148.787,Z 325.12,A -85,B 0,C 180,E1 -26784.572,E2 -26784.572} C_VEL
LIN {X 0,Y 153.578,Z 313.669,A -85,B 0,C 180,E1 -26786.044,E2 -26786.044} C_VEL
LIN {X 0,Y 155.798,Z 307.406,A -85,B 0,C 180,E1 -26786.628,E2 -26786.628} C_VEL
LIN {X 0,Y 157.128,Z 301.924,A -85,B 0,C 180,E1 -26787.283,E2 -26787.283} C_VEL
LIN {X 0,Y 158.034,Z 289.365,A -85,B 0,C 180,E1 -26789.419,E2 -26789.419} C_VEL
LIN {X 0,Y 158.355,Z 281.929,A -85,B 0,C 180,E1 -26790.389,E2 -26790.389} C_VEL
LIN {X 0,Y 158.685,Z 278.067,A -85,B 0,C 180,E1 -26790.641,E2 -26790.641} C_VEL
LIN {X 0,Y 159.713,Z 266.896,A -85,B 0,C 180,E1 -26791.05,E2 -26791.05} C_VEL
LIN {X 0,Y 156.979,Z 258.476,A -85,B 0,C 180,E1 -26794.009,E2 -26794.009} C_VEL
LIN {X 0,Y 154.347,Z 251.107,A -85,B 0,C 180,E1 -26797.252,E2 -26797.252} C_VEL
LIN {X 0,Y 152.056,Z 245.548,A -85,B 0,C 180,E1 -26800.525,E2 -26800.525} C_VEL
LIN {X 0,Y 150.647,Z 243.109,A -85,B 0,C 180,E1 -26802.764,E2 -26802.764} C_VEL
LIN {X 0,Y 149.322,Z 240.615,A -85,B 0,C 180,E1 -26805.309,E2 -26805.309} C_VEL
LIN {X 0,Y 147.426,Z 237.059,A -85,B 0,C 180,E1 -26810.435,E2 -26810.435} C_VEL
LIN {X 0,Y 147.111,Z 236.331,A -85,B 0,C 180,E1 -26811.76,E2 -26811.76} C_VEL
LIN {X 0,Y 146.484,Z 235.519,A -85,B 0,C 180,E1 -26820,E2 -26820} C_VEL
LIN {X 0,Y 147.388,Z 236.607,A -85,B 0,C 180,E1 -26824.958,E2 -26824.958} C_VEL
LIN {X 0,Y 148.914,Z 240.045,A -85,B 0,C 180,E1 -26829.508,E2 -26829.508} C_VEL
LIN {X 0,Y 149.721,Z 241.267,A -85,B 0,C 180,E1 -26831.165,E2 -26831.165} C_VEL
LIN {X 0,Y 152.178,Z 245.674,A -85,B 0,C 180,E1 -26835.314,E2 -26835.314} C_VEL
LIN {X 0,Y 154.933,Z 250.726,A -85,B 0,C 180,E1 -26838.943,E2 -26838.943} C_VEL
LIN {X 0,Y 158.272,Z 257.576,A -85,B 0,C 180,E1 -26842.606,E2 -26842.606} C_VEL
LIN {X 0,Y 160.247,Z 261.935,A -85,B 0,C 180,E1 -26844.518,E2 -26844.518} C_VEL
LIN {X 0,Y 158.285,Z 278.882,A -85,B 0,C 180,E1 -26845.144,E2 -26845.144} C_VEL
LIN {X 0,Y 155.722,Z 291.215,A -85,B 0,C 180,E1 -26845.907,E2 -26845.907} C_VEL
LIN {X 0,Y 151.891,Z 303.934,A -85,B 0,C 180,E1 -26847.06,E2 -26847.06} C_VEL
LIN {X 0,Y 147.042,Z 316.131,A -85,B 0,C 180,E1 -26848.596,E2 -26848.596} C_VEL
LIN {X 0,Y 141.709,Z 326.88,A -85,B 0,C 180,E1 -26850.488,E2 -26850.488} C_VEL
LIN {X 0,Y 135.796,Z 336.68,A -85,B 0,C 180,E1 -26852.75,E2 -26852.75} C_VEL
LIN {X 0,Y 129.446,Z 345.576,A -85,B 0,C 180,E1 -26855.469,E2 -26855.469} C_VEL
LIN {X 0,Y 122.693,Z 353.796,A -85,B 0,C 180,E1 -26858.911,E2 -26858.911} C_VEL
LIN {X 0,Y 115.789,Z 361.099,A -85,B 0,C 180,E1 -26863.247,E2 -26863.247} C_VEL
LIN {X 0,Y 109.703,Z 366.587,A -85,B 0,C 180,E1 -26867.723,E2 -26867.723} C_VEL
LIN {X 0,Y 104.355,Z 370.872,A -85,B 0,C 180,E1 -26872.687,E2 -26872.687} C_VEL
LIN {X 0,Y 100.723,Z 373.479,A -85,B 0,C 180,E1 -26876.858,E2 -26876.858} C_VEL
LIN {X 0,Y 96.163,Z 376.3,A -85,B 0,C 180,E1 -26883.987,E2 -26883.987} C_VEL
LIN {X 0,Y 92.843,Z 377.818,A -85,B 0,C 180,E1 -26892.371,E2 -26892.371} C_VEL
LIN {X 0,Y 91.896,Z 377.984,A -85,B 0,C 180,E1 -26896.732,E2 -26896.732} C_VEL
LIN {X 0,Y 91.383,Z 377.725,A -85,B 0,C 180,E1 -26901.148,E2 -26901.148} C_VEL
LIN {X 0,Y 91.368,Z 376.188,A -85,B 0,C 180,E1 -26909.55,E2 -26909.55} C_VEL
LIN {X 0,Y 91.944,Z 374.66,A -85,B 0,C 180,E1 -26914.38,E2 -26914.38} C_VEL
LIN {X 0,Y 93.589,Z 371.726,A -85,B 0,C 180,E1 -26920.816,E2 -26920.816} C_VEL
LIN {X 0,Y 96.074,Z 367.771,A -85,B 0,C 180,E1 -26927.01,E2 -26927.01} C_VEL
LIN {X 0,Y 100.227,Z 361.675,A -85,B 0,C 180,E1 -26933.774,E2 -26933.774} C_VEL
LIN {X 0,Y 104.812,Z 354.802,A -85,B 0,C 180,E1 -26939.293,E2 -26939.293} C_VEL
LIN {X 0,Y 109.843,Z 346.8,A -85,B 0,C 180,E1 -26944.04,E2 -26944.04} C_VEL
LIN {X 0,Y 114.7,Z 338.327,A -85,B 0,C 180,E1 -26947.783,E2 -26947.783} C_VEL
LIN {X 0,Y 119.962,Z 327.87,A -85,B 0,C 180,E1 -26951.225,E2 -26951.225} C_VEL
LIN {X 0,Y 124.337,Z 317.524,A -85,B 0,C 180,E1 -26953.817,E2 -26953.817} C_VEL
LIN {X 0,Y 128.386,Z 306.151,A -85,B 0,C 180,E1 -26955.924,E2 -26955.924} C_VEL
LIN {X 0,Y 131.664,Z 294.389,A -85,B 0,C 180,E1 -26957.496,E2 -26957.496} C_VEL
LIN {X 0,Y 134.353,Z 280.572,A -85,B 0,C 180,E1 -26958.796,E2 -26958.796} C_VEL
LIN {X 0,Y 135.859,Z 267.887,A -85,B 0,C 180,E1 -26959.51,E2 -26959.51} C_VEL
LIN {X 0,Y 137.953,Z 242.285,A -85,B 0,C 180,E1 -26960.534,E2 -26960.534} C_VEL
LIN {X 0,Y 134.662,Z 235.181,A -85,B 0,C 180,E1 -26963.124,E2 -26963.124} C_VEL
LIN {X 0,Y 130.754,Z 227.832,A -85,B 0,C 180,E1 -26966.523,E2 -26966.523} C_VEL
LIN {X 0,Y 127.119,Z 221.69,A -85,B 0,C 180,E1 -26970.159,E2 -26970.159} C_VEL
LIN {X 0,Y 125.011,Z 218.393,A -85,B 0,C 180,E1 -26972.567,E2 -26972.567} C_VEL
LIN {X 0,Y 122.971,Z 215.169,A -85,B 0,C 180,E1 -26975.225,E2 -26975.225} C_VEL
LIN {X 0,Y 120.376,Z 211.196,A -85,B 0,C 180,E1 -26979.272,E2 -26979.272} C_VEL
LIN {X 0,Y 117.763,Z 208.083,A -85,B 0,C 180,E1 -26984.587,E2 -26984.587} C_VEL
LIN {X 0,Y 116.975,Z 206.006,A -85,B 0,C 180,E1 -26987.15,E2 -26987.15} C_VEL
LIN {X 0,Y 115.352,Z 204.736,A -85,B 0,C 180,E1 -26996.507,E2 -26996.507} C_VEL
LIN {X 0,Y 115.573,Z 204.782,A -85,B 0,C 180,E1 -27000.871,E2 -27000.871} C_VEL
LIN {X 0,Y 117.167,Z 206.219,A -85,B 0,C 180,E1 -27007.837,E2 -27007.837} C_VEL
LIN {X 0,Y 118.506,Z 209.208,A -85,B 0,C 180,E1 -27011.6,E2 -27011.6} C_VEL
LIN {X 0,Y 120.521,Z 211.418,A -85,B 0,C 180,E1 -27015.375,E2 -27015.375} C_VEL
LIN {X 0,Y 122.839,Z 215.013,A -85,B 0,C 180,E1 -27018.989,E2 -27018.989} C_VEL
LIN {X 0,Y 124.19,Z 217.076,A -85,B 0,C 180,E1 -27020.794,E2 -27020.794} C_VEL
LIN {X 0,Y 126.512,Z 220.676,A -85,B 0,C 180,E1 -27023.56,E2 -27023.56} C_VEL
LIN {X 0,Y 129.918,Z 226.195,A -85,B 0,C 180,E1 -27027.062,E2 -27027.062} C_VEL
LIN {X 0,Y 132.715,Z 232.729,A -85,B 0,C 180,E1 -27029.758,E2 -27029.758} C_VEL
LIN {X 0,Y 136.098,Z 242.32,A -85,B 0,C 180,E1 -27032.793,E2 -27032.793} C_VEL
LIN {X 0,Y 137.474,Z 247.057,A -85,B 0,C 180,E1 -27033.997,E2 -27033.997} C_VEL
LIN {X 0,Y 137.215,Z 252.275,A -85,B 0,C 180,E1 -27034.299,E2 -27034.299} C_VEL
LIN {X 0,Y 134.49,Z 282.692,A -85,B 0,C 180,E1 -27035.544,E2 -27035.544} C_VEL
LIN {X 0,Y 132.156,Z 296.164,A -85,B 0,C 180,E1 -27036.503,E2 -27036.503} C_VEL
LIN {X 0,Y 129.041,Z 308.499,A -85,B 0,C 180,E1 -27037.847,E2 -27037.847} C_VEL
LIN {X 0,Y 125.271,Z 319.651,A -85,B 0,C 180,E1 -27039.525,E2 -27039.525} C_VEL
LIN {X 0,Y 120.424,Z 331.26,A -85,B 0,C 180,E1 -27041.924,E2 -27041.924} C_VEL
LIN {X 0,Y 115.33,Z 341.722,A -85,B 0,C 180,E1 -27044.9,E2 -27044.9} C_VEL
LIN {X 0,Y 110.584,Z 350.272,A -85,B 0,C 180,E1 -27048.146,E2 -27048.146} C_VEL
LIN {X 0,Y 105.871,Z 358.165,A -85,B 0,C 180,E1 -27052.123,E2 -27052.123} C_VEL
LIN {X 0,Y 101.011,Z 365.874,A -85,B 0,C 180,E1 -27057.374,E2 -27057.374} C_VEL
LIN {X 0,Y 96.389,Z 372.984,A -85,B 0,C 180,E1 -27064.062,E2 -27064.062} C_VEL
LIN {X 0,Y 93.451,Z 377.7,A -85,B 0,C 180,E1 -27070.224,E2 -27070.224} C_VEL
LIN {X 0,Y 91.78,Z 381.307,A -85,B 0,C 180,E1 -27076.723,E2 -27076.723} C_VEL
LIN {X 0,Y 91.205,Z 383.149,A -85,B 0,C 180,E1 -27081.139,E2 -27081.139} C_VEL
LIN {X 0,Y 91.054,Z 384.529,A -85,B 0,C 180,E1 -27085.577,E2 -27085.577} C_VEL
LIN {X 0,Y 91.218,Z 385.505,A -85,B 0,C 180,E1 -27090.004,E2 -27090.004} C_VEL
LIN {X 0,Y 91.052,Z 386.052,A -85,B 0,C 180,E1 -27094.431,E2 -27094.431} C_VEL
LIN {X 0,Y 91.195,Z 386.185,A -85,B 0,C 180,E1 -27098.87,E2 -27098.87} C_VEL
LIN {X 0,Y 92.895,Z 385.23,A -85,B 0,C 180,E1 -27107.619,E2 -27107.619} C_VEL
LIN {X 0,Y 94.462,Z 384.179,A -85,B 0,C 180,E1 -27111.843,E2 -27111.843} C_VEL
LIN {X 0,Y 96.639,Z 382.728,A -85,B 0,C 180,E1 -27115.875,E2 -27115.875} C_VEL
LIN {X 0,Y 100.676,Z 379.731,A -85,B 0,C 180,E1 -27121.575,E2 -27121.575} C_VEL
LIN {X 0,Y 106.509,Z 374.89,A -85,B 0,C 180,E1 -27127.645,E2 -27127.645} C_VEL
LIN {X 0,Y 113.358,Z 368.528,A -85,B 0,C 180,E1 -27133.002,E2 -27133.002} C_VEL
LIN {X 0,Y 120.07,Z 361.61,A -85,B 0,C 180,E1 -27137.029,E2 -27137.029} C_VEL
LIN {X 0,Y 127.366,Z 352.972,A -85,B 0,C 180,E1 -27140.584,E2 -27140.584} C_VEL
LIN {X 0,Y 133.864,Z 344.133,A -85,B 0,C 180,E1 -27143.195,E2 -27143.195} C_VEL
LIN {X 0,Y 140.609,Z 333.268,A -85,B 0,C 180,E1 -27145.563,E2 -27145.563} C_VEL
LIN {X 0,Y 146.233,Z 322.319,A -85,B 0,C 180,E1 -27147.255,E2 -27147.255} C_VEL
LIN {X 0,Y 151.188,Z 310.062,A -85,B 0,C 180,E1 -27148.671,E2 -27148.671} C_VEL
LIN {X 0,Y 154.794,Z 298.489,A -85,B 0,C 180,E1 -27149.618,E2 -27149.618} C_VEL
LIN {X 0,Y 157.665,Z 285.262,A -85,B 0,C 180,E1 -27150.364,E2 -27150.364} C_VEL
LIN {X 0,Y 158.685,Z 278.067,A -85,B 0,C 180,E1 -27150.641,E2 -27150.641} C_VEL
LIN {X 0,Y 158.714,Z 274.991,A -85,B 0,C 180,E1 -27150.971,E2 -27150.971} C_VEL
LIN {X 0,Y 157.956,Z 271.284,A -85,B 0,C 180,E1 -27151.913,E2 -27151.913} C_VEL
LIN {X 0,Y 157.298,Z 269.511,A -85,B 0,C 180,E1 -27152.595,E2 -27152.595} C_VEL
LIN {X 0,Y 154.254,Z 262.877,A -85,B 0,C 180,E1 -27155.865,E2 -27155.865} C_VEL
LIN {X 0,Y 152.054,Z 256.231,A -85,B 0,C 180,E1 -27158.938,E2 -27158.938} C_VEL
LIN {X 0,Y 150.336,Z 251.717,A -85,B 0,C 180,E1 -27161.694,E2 -27161.694} C_VEL
LIN {X 0,Y 148.04,Z 247.349,A -85,B 0,C 180,E1 -27166.088,E2 -27166.088} C_VEL
LIN {X 0,Y 146.25,Z 243.409,A -85,B 0,C 180,E1 -27171.711,E2 -27171.711} C_VEL
LIN {X 0,Y 145.614,Z 242.587,A -85,B 0,C 180,E1 -27180,E2 -27180} C_VEL
LIN {X 0,Y 146.371,Z 243.62,A -85,B 0,C 180,E1 -27184.475,E2 -27184.475} C_VEL
LIN {X 0,Y 147.887,Z 247.06,A -85,B 0,C 180,E1 -27189.23,E2 -27189.23} C_VEL
LIN {X 0,Y 148.567,Z 248.339,A -85,B 0,C 180,E1 -27190.735,E2 -27190.735} C_VEL
LIN {X 0,Y 150.525,Z 252.013,A -85,B 0,C 180,E1 -27194.276,E2 -27194.276} C_VEL
LIN {X 0,Y 153.105,Z 257.078,A -85,B 0,C 180,E1 -27197.964,E2 -27197.964} C_VEL
LIN {X 0,Y 156.469,Z 264.557,A -85,B 0,C 180,E1 -27201.919,E2 -27201.919} C_VEL
LIN {X 0,Y 156.82,Z 265.415,A -85,B 0,C 180,E1 -27202.296,E2 -27202.296} C_VEL
LIN {X 0,Y 154.982,Z 280.061,A -85,B 0,C 180,E1 -27202.869,E2 -27202.869} C_VEL
LIN {X 0,Y 152.131,Z 292.78,A -85,B 0,C 180,E1 -27203.663,E2 -27203.663} C_VEL
LIN {X 0,Y 148.007,Z 305.71,A -85,B 0,C 180,E1 -27204.843,E2 -27204.843} C_VEL
LIN {X 0,Y 143.081,Z 317.367,A -85,B 0,C 180,E1 -27206.315,E2 -27206.315} C_VEL
LIN {X 0,Y 137.526,Z 327.958,A -85,B 0,C 180,E1 -27208.168,E2 -27208.168} C_VEL
LIN {X 0,Y 132.066,Z 336.653,A -85,B 0,C 180,E1 -27210.141,E2 -27210.141} C_VEL
LIN {X 0,Y 125.425,Z 345.607,A -85,B 0,C 180,E1 -27212.802,E2 -27212.802} C_VEL
LIN {X 0,Y 118.124,Z 354.107,A -85,B 0,C 180,E1 -27216.323,E2 -27216.323} C_VEL
LIN {X 0,Y 111.006,Z 361.243,A -85,B 0,C 180,E1 -27220.555,E2 -27220.555} C_VEL
LIN {X 0,Y 104.507,Z 366.767,A -85,B 0,C 180,E1 -27225.076,E2 -27225.076} C_VEL
LIN {X 0,Y 98.753,Z 371.086,A -85,B 0,C 180,E1 -27230.166,E2 -27230.166} C_VEL
LIN {X 0,Y 94.452,Z 373.937,A -85,B 0,C 180,E1 -27234.935,E2 -27234.935} C_VEL
LIN {X 0,Y 89.789,Z 376.575,A -85,B 0,C 180,E1 -27241.985,E2 -27241.985} C_VEL
LIN {X 0,Y 86.064,Z 378.121,A -85,B 0,C 180,E1 -27250.931,E2 -27250.931} C_VEL
LIN {X 0,Y 84.959,Z 378.312,A -85,B 0,C 180,E1 -27255.627,E2 -27255.627} C_VEL
LIN {X 0,Y 84.354,Z 378.071,A -85,B 0,C 180,E1 -27260.404,E2 -27260.404} C_VEL
LIN {X 0,Y 84.13,Z 377.449,A -85,B 0,C 180,E1 -27265.204,E2 -27265.204} C_VEL
LIN {X 0,Y 84.34,Z 376.331,A -85,B 0,C 180,E1 -27270.496,E2 -27270.496} C_VEL
LIN {X 0,Y 84.877,Z 375.059,A -85,B 0,C 180,E1 -27274.745,E2 -27274.745} C_VEL
LIN {X 0,Y 86.652,Z 372.15,A -85,B 0,C 180,E1 -27281.694,E2 -27281.694} C_VEL
LIN {X 0,Y 89.336,Z 368.226,A -85,B 0,C 180,E1 -27288.337,E2 -27288.337} C_VEL
LIN {X 0,Y 93.081,Z 363.169,A -85,B 0,C 180,E1 -27294.532,E2 -27294.532} C_VEL
LIN {X 0,Y 97.668,Z 356.805,A -85,B 0,C 180,E1 -27300.241,E2 -27300.241} C_VEL
LIN {X 0,Y 103.096,Z 348.866,A -85,B 0,C 180,E1 -27305.406,E2 -27305.406} C_VEL
LIN {X 0,Y 108.138,Z 340.774,A -85,B 0,C 180,E1 -27309.316,E2 -27309.316} C_VEL
LIN {X 0,Y 113.597,Z 330.906,A -85,B 0,C 180,E1 -27312.881,E2 -27312.881} C_VEL
LIN {X 0,Y 118.791,Z 319.768,A -85,B 0,C 180,E1 -27315.83,E2 -27315.83} C_VEL
LIN {X 0,Y 122.993,Z 308.865,A -85,B 0,C 180,E1 -27317.968,E2 -27317.968} C_VEL
LIN {X 0,Y 126.676,Z 296.808,A -85,B 0,C 180,E1 -27319.711,E2 -27319.711} C_VEL
LIN {X 0,Y 129.617,Z 283.579,A -85,B 0,C 180,E1 -27321.011,E2 -27321.011} C_VEL
LIN {X 0,Y 131.446,Z 270.071,A -85,B 0,C 180,E1 -27321.855,E2 -27321.855} C_VEL
LIN {X 0,Y 133.543,Z 244.924,A -85,B 0,C 180,E1 -27322.917,E2 -27322.917} C_VEL
LIN {X 0,Y 129.681,Z 236.623,A -85,B 0,C 180,E1 -27326.387,E2 -27326.387} C_VEL
LIN {X 0,Y 126.213,Z 230.187,A -85,B 0,C 180,E1 -27329.923,E2 -27329.923} C_VEL
LIN {X 0,Y 123.192,Z 224.952,A -85,B 0,C 180,E1 -27333.533,E2 -27333.533} C_VEL
LIN {X 0,Y 120.953,Z 221.352,A -85,B 0,C 180,E1 -27336.681,E2 -27336.681} C_VEL
LIN {X 0,Y 118.611,Z 217.555,A -85,B 0,C 180,E1 -27340.742,E2 -27340.742} C_VEL
LIN {X 0,Y 116.501,Z 214.783,A -85,B 0,C 180,E1 -27345.546,E2 -27345.546} C_VEL
LIN {X 0,Y 115.795,Z 212.918,A -85,B 0,C 180,E1 -27348.08,E2 -27348.08} C_VEL
LIN {X 0,Y 114.486,Z 211.784,A -85,B 0,C 180,E1 -27356.48,E2 -27356.48} C_VEL
LIN {X 0,Y 114.67,Z 211.794,A -85,B 0,C 180,E1 -27360.548,E2 -27360.548} C_VEL
LIN {X 0,Y 115.988,Z 213.098,A -85,B 0,C 180,E1 -27366.96,E2 -27366.96} C_VEL
LIN {X 0,Y 117.394,Z 216.196,A -85,B 0,C 180,E1 -27371.164,E2 -27371.164} C_VEL
LIN {X 0,Y 118.981,Z 218.067,A -85,B 0,C 180,E1 -27374.348,E2 -27374.348} C_VEL
LIN {X 0,Y 121.381,Z 221.841,A -85,B 0,C 180,E1 -27378.323,E2 -27378.323} C_VEL
LIN {X 0,Y 124.515,Z 227.136,A -85,B 0,C 180,E1 -27382.504,E2 -27382.504} C_VEL
LIN {X 0,Y 127.594,Z 232.564,A -85,B 0,C 180,E1 -27385.926,E2 -27385.926} C_VEL
LIN {X 0,Y 130.607,Z 240.743,A -85,B 0,C 180,E1 -27389.104,E2 -27389.104} C_VEL
LIN {X 0,Y 133.301,Z 249.437,A -85,B 0,C 180,E1 -27391.742,E2 -27391.742} C_VEL
LIN {X 0,Y 130.227,Z 282.504,A -85,B 0,C 180,E1 -27393.089,E2 -27393.089} C_VEL
LIN {X 0,Y 127.804,Z 295.925,A -85,B 0,C 180,E1 -27394.035,E2 -27394.035} C_VEL
LIN {X 0,Y 124.461,Z 308.516,A -85,B 0,C 180,E1 -27395.394,E2 -27395.394} C_VEL
LIN {X 0,Y 120.231,Z 320.385,A -85,B 0,C 180,E1 -27397.215,E2 -27397.215} C_VEL
LIN {X 0,Y 115.176,Z 331.801,A -85,B 0,C 180,E1 -27399.618,E2 -27399.618} C_VEL
LIN {X 0,Y 109.832,Z 342.099,A -85,B 0,C 180,E1 -27402.625,E2 -27402.625} C_VEL
LIN {X 0,Y 104.301,Z 351.344,A -85,B 0,C 180,E1 -27406.323,E2 -27406.323} C_VEL
LIN {X 0,Y 98.452,Z 360.359,A -85,B 0,C 180,E1 -27411.352,E2 -27411.352} C_VEL
LIN {X 0,Y 94.304,Z 366.493,A -85,B 0,C 180,E1 -27416.023,E2 -27416.023} C_VEL
LIN {X 0,Y 90.025,Z 372.507,A -85,B 0,C 180,E1 -27422.075,E2 -27422.075} C_VEL
LIN {X 0,Y 86.758,Z 377.254,A -85,B 0,C 180,E1 -27428.626,E2 -27428.626} C_VEL
LIN {X 0,Y 84.832,Z 380.891,A -85,B 0,C 180,E1 -27435.614,E2 -27435.614} C_VEL
LIN {X 0,Y 84.17,Z 382.76,A -85,B 0,C 180,E1 -27440.391,E2 -27440.391} C_VEL
LIN {X 0,Y 83.972,Z 384.158,A -85,B 0,C 180,E1 -27445.204,E2 -27445.204} C_VEL
LIN {X 0,Y 84.133,Z 385.148,A -85,B 0,C 180,E1 -27450.004,E2 -27450.004} C_VEL
LIN {X 0,Y 83.971,Z 385.707,A -85,B 0,C 180,E1 -27454.805,E2 -27454.805} C_VEL
LIN {X 0,Y 84.164,Z 385.864,A -85,B 0,C 180,E1 -27459.618,E2 -27459.618} C_VEL
LIN {X 0,Y 86.134,Z 384.939,A -85,B 0,C 180,E1 -27469.053,E2 -27469.053} C_VEL
LIN {X 0,Y 87.878,Z 383.9,A -85,B 0,C 180,E1 -27473.574,E2 -27473.574} C_VEL
LIN {X 0,Y 90.274,Z 382.472,A -85,B 0,C 180,E1 -27477.851,E2 -27477.851} C_VEL
LIN {X 0,Y 94.684,Z 379.498,A -85,B 0,C 180,E1 -27483.832,E2 -27483.832} C_VEL
LIN {X 0,Y 100.392,Z 375.163,A -85,B 0,C 180,E1 -27489.641,E2 -27489.641} C_VEL
LIN {X 0,Y 107.132,Z 369.387,A -85,B 0,C 180,E1 -27494.851,E2 -27494.851} C_VEL
LIN {X 0,Y 114.102,Z 362.73,A -85,B 0,C 180,E1 -27498.988,E2 -27498.988} C_VEL
LIN {X 0,Y 121.687,Z 354.488,A -85,B 0,C 180,E1 -27502.577,E2 -27502.577} C_VEL
LIN {X 0,Y 128.332,Z 346.069,A -85,B 0,C 180,E1 -27505.235,E2 -27505.235} C_VEL
LIN {X 0,Y 135.314,Z 335.69,A -85,B 0,C 180,E1 -27507.569,E2 -27507.569} C_VEL
LIN {X 0,Y 141.8,Z 324.009,A -85,B 0,C 180,E1 -27509.45,E2 -27509.45} C_VEL
LIN {X 0,Y 146.859,Z 312.4,A -85,B 0,C 180,E1 -27510.855,E2 -27510.855} C_VEL
LIN {X 0,Y 150.615,Z 301.637,A -85,B 0,C 180,E1 -27511.736,E2 -27511.736} C_VEL
LIN {X 0,Y 153.837,Z 288.668,A -85,B 0,C 180,E1 -27512.53,E2 -27512.53} C_VEL
LIN {X 0,Y 155.866,Z 275.539,A -85,B 0,C 180,E1 -27513.039,E2 -27513.039} C_VEL
LIN {X 0,Y 156.349,Z 269.741,A -85,B 0,C 180,E1 -27513.288,E2 -27513.288} C_VEL
LIN {X 0,Y 154.254,Z 262.877,A -85,B 0,C 180,E1 -27515.865,E2 -27515.865} C_VEL
LIN {X 0,Y 152.79,Z 259.8,A -85,B 0,C 180,E1 -27517.67,E2 -27517.67} C_VEL
LIN {X 0,Y 151.179,Z 257.791,A -85,B 0,C 180,E1 -27519.697,E2 -27519.697} C_VEL
LIN {X 0,Y 146.663,Z 253.887,A -85,B 0,C 180,E1 -27527.182,E2 -27527.182} C_VEL
LIN {X 0,Y 145.226,Z 250.355,A -85,B 0,C 180,E1 -27532.353,E2 -27532.353} C_VEL
LIN {X 0,Y 144.746,Z 249.651,A -85,B 0,C 180,E1 -27540,E2 -27540} C_VEL
LIN {X 0,Y 145.402,Z 250.712,A -85,B 0,C 180,E1 -27544.158,E2 -27544.158} C_VEL
LIN {X 0,Y 146.865,Z 254.068,A -85,B 0,C 180,E1 -27548.948,E2 -27548.948} C_VEL
LIN {X 0,Y 149.062,Z 258.672,A -85,B 0,C 180,E1 -27553.462,E2 -27553.462} C_VEL
LIN {X 0,Y 151.263,Z 263.352,A -85,B 0,C 180,E1 -27556.882,E2 -27556.882} C_VEL
LIN {X 0,Y 153.655,Z 268.974,A -85,B 0,C 180,E1 -27560.002,E2 -27560.002} C_VEL
LIN {X 0,Y 151.664,Z 282.437,A -85,B 0,C 180,E1 -27560.564,E2 -27560.564} C_VEL
LIN {X 0,Y 148.47,Z 295.458,A -85,B 0,C 180,E1 -27561.4,E2 -27561.4} C_VEL
LIN {X 0,Y 144.491,Z 307.063,A -85,B 0,C 180,E1 -27562.454,E2 -27562.454} C_VEL
LIN {X 0,Y 139.462,Z 318.344,A -85,B 0,C 180,E1 -27563.866,E2 -27563.866} C_VEL
LIN {X 0,Y 133.58,Z 329.035,A -85,B 0,C 180,E1 -27565.707,E2 -27565.707} C_VEL
LIN {X 0,Y 127.234,Z 338.58,A -85,B 0,C 180,E1 -27567.893,E2 -27567.893} C_VEL
LIN {X 0,Y 120.347,Z 347.266,A -85,B 0,C 180,E1 -27570.525,E2 -27570.525} C_VEL
LIN {X 0,Y 113.564,Z 354.673,A -85,B 0,C 180,E1 -27573.653,E2 -27573.653} C_VEL
LIN {X 0,Y 106.477,Z 361.388,A -85,B 0,C 180,E1 -27577.617,E2 -27577.617} C_VEL
LIN {X 0,Y 99.567,Z 366.947,A -85,B 0,C 180,E1 -27582.166,E2 -27582.166} C_VEL
LIN {X 0,Y 93.356,Z 371.3,A -85,B 0,C 180,E1 -27587.344,E2 -27587.344} C_VEL
LIN {X 0,Y 88.248,Z 374.409,A -85,B 0,C 180,E1 -27592.789,E2 -27592.789} C_VEL
LIN {X 0,Y 83.546,Z 376.85,A -85,B 0,C 180,E1 -27599.682,E2 -27599.682} C_VEL
LIN {X 0,Y 79.335,Z 378.426,A -85,B 0,C 180,E1 -27609.242,E2 -27609.242} C_VEL
LIN {X 0,Y 78.072,Z 378.635,A -85,B 0,C 180,E1 -27614.328,E2 -27614.328} C_VEL
LIN {X 0,Y 77.332,Z 378.418,A -85,B 0,C 180,E1 -27619.523,E2 -27619.523} C_VEL
LIN {X 0,Y 77.054,Z 377.809,A -85,B 0,C 180,E1 -27624.762,E2 -27624.762} C_VEL
LIN {X 0,Y 77.333,Z 376.503,A -85,B 0,C 180,E1 -27631.426,E2 -27631.426} C_VEL
LIN {X 0,Y 78.944,Z 373.629,A -85,B 0,C 180,E1 -27640.251,E2 -27640.251} C_VEL
LIN {X 0,Y 81.574,Z 370.088,A -85,B 0,C 180,E1 -27647.545,E2 -27647.545} C_VEL
LIN {X 0,Y 85.2,Z 365.456,A -85,B 0,C 180,E1 -27654.353,E2 -27654.353} C_VEL
LIN {X 0,Y 90.738,Z 358.478,A -85,B 0,C 180,E1 -27661.516,E2 -27661.516} C_VEL
LIN {X 0,Y 96.41,Z 350.919,A -85,B 0,C 180,E1 -27666.965,E2 -27666.965} C_VEL
LIN {X 0,Y 102.775,Z 341.415,A -85,B 0,C 180,E1 -27671.81,E2 -27671.81} C_VEL
LIN {X 0,Y 108.525,Z 331.611,A -85,B 0,C 180,E1 -27675.421,E2 -27675.421} C_VEL
LIN {X 0,Y 113.996,Z 320.599,A -85,B 0,C 180,E1 -27678.37,E2 -27678.37} C_VEL
LIN {X 0,Y 118.396,Z 309.817,A -85,B 0,C 180,E1 -27680.499,E2 -27680.499} C_VEL
LIN {X 0,Y 122.251,Z 297.934,A -85,B 0,C 180,E1 -27682.223,E2 -27682.223} C_VEL
LIN {X 0,Y 125.274,Z 285.309,A -85,B 0,C 180,E1 -27683.514,E2 -27683.514} C_VEL
LIN {X 0,Y 127.298,Z 271.843,A -85,B 0,C 180,E1 -27684.38,E2 -27684.38} C_VEL
LIN {X 0,Y 129.471,Z 247.868,A -85,B 0,C 180,E1 -27685.361,E2 -27685.361} C_VEL
LIN {X 0,Y 126.036,Z 240.323,A -85,B 0,C 180,E1 -27688.86,E2 -27688.86} C_VEL
LIN {X 0,Y 122.377,Z 233.332,A -85,B 0,C 180,E1 -27693.204,E2 -27693.204} C_VEL
LIN {X 0,Y 119.418,Z 228.05,A -85,B 0,C 180,E1 -27697.54,E2 -27697.54} C_VEL
LIN {X 0,Y 117.111,Z 224.2,A -85,B 0,C 180,E1 -27701.855,E2 -27701.855} C_VEL
LIN {X 0,Y 115.14,Z 221.154,A -85,B 0,C 180,E1 -27706.993,E2 -27706.993} C_VEL
LIN {X 0,Y 114.696,Z 219.849,A -85,B 0,C 180,E1 -27708.85,E2 -27708.85} C_VEL
LIN {X 0,Y 113.62,Z 218.84,A -85,B 0,C 180,E1 -27716.453,E2 -27716.453} C_VEL
LIN {X 0,Y 113.86,Z 218.946,A -85,B 0,C 180,E1 -27721.105,E2 -27721.105} C_VEL
LIN {X 0,Y 114.858,Z 220.008,A -85,B 0,C 180,E1 -27726.147,E2 -27726.147} C_VEL
LIN {X 0,Y 116.401,Z 223.334,A -85,B 0,C 180,E1 -27730.986,E2 -27730.986} C_VEL
LIN {X 0,Y 117.574,Z 224.949,A -85,B 0,C 180,E1 -27733.503,E2 -27733.503} C_VEL
LIN {X 0,Y 120.119,Z 229.27,A -85,B 0,C 180,E1 -27737.971,E2 -27737.971} C_VEL
LIN {X 0,Y 123.272,Z 234.782,A -85,B 0,C 180,E1 -27742.302,E2 -27742.302} C_VEL
LIN {X 0,Y 125.161,Z 238.777,A -85,B 0,C 180,E1 -27744.588,E2 -27744.588} C_VEL
LIN {X 0,Y 127.941,Z 247.236,A -85,B 0,C 180,E1 -27747.836,E2 -27747.836} C_VEL
LIN {X 0,Y 129.198,Z 251.632,A -85,B 0,C 180,E1 -27749.222,E2 -27749.222} C_VEL
LIN {X 0,Y 126.313,Z 281.772,A -85,B 0,C 180,E1 -27750.452,E2 -27750.452} C_VEL
LIN {X 0,Y 123.857,Z 294.976,A -85,B 0,C 180,E1 -27751.335,E2 -27751.335} C_VEL
LIN {X 0,Y 120.485,Z 307.469,A -85,B 0,C 180,E1 -27752.639,E2 -27752.639} C_VEL
LIN {X 0,Y 116.054,Z 319.521,A -85,B 0,C 180,E1 -27754.408,E2 -27754.408} C_VEL
LIN {X 0,Y 110.763,Z 331.036,A -85,B 0,C 180,E1 -27756.774,E2 -27756.774} C_VEL
LIN {X 0,Y 105.151,Z 341.426,A -85,B 0,C 180,E1 -27759.776,E2 -27759.776} C_VEL
LIN {X 0,Y 99.27,Z 350.743,A -85,B 0,C 180,E1 -27763.482,E2 -27763.482} C_VEL
LIN {X 0,Y 92.875,Z 359.937,A -85,B 0,C 180,E1 -27768.688,E2 -27768.688} C_VEL
LIN {X 0,Y 88.403,Z 365.982,A -85,B 0,C 180,E1 -27773.417,E2 -27773.417} C_VEL
LIN {X 0,Y 83.766,Z 372.027,A -85,B 0,C 180,E1 -27779.78,E2 -27779.78} C_VEL
LIN {X 0,Y 80.154,Z 376.809,A -85,B 0,C 180,E1 -27786.766,E2 -27786.766} C_VEL
LIN {X 0,Y 77.935,Z 380.476,A -85,B 0,C 180,E1 -27794.309,E2 -27794.309} C_VEL
LIN {X 0,Y 77.137,Z 382.368,A -85,B 0,C 180,E1 -27799.506,E2 -27799.506} C_VEL
LIN {X 0,Y 76.886,Z 383.787,A -85,B 0,C 180,E1 -27804.76,E2 -27804.76} C_VEL
LIN {X 0,Y 77.05,Z 384.792,A -85,B 0,C 180,E1 -27810.005,E2 -27810.005} C_VEL
LIN {X 0,Y 76.885,Z 385.363,A -85,B 0,C 180,E1 -27815.249,E2 -27815.249} C_VEL
LIN {X 0,Y 77.166,Z 385.54,A -85,B 0,C 180,E1 -27820.5,E2 -27820.5} C_VEL
LIN {X 0,Y 79.423,Z 384.647,A -85,B 0,C 180,E1 -27830.734,E2 -27830.734} C_VEL
LIN {X 0,Y 81.391,Z 383.623,A -85,B 0,C 180,E1 -27835.583,E2 -27835.583} C_VEL
LIN {X 0,Y 84.035,Z 382.213,A -85,B 0,C 180,E1 -27840.123,E2 -27840.123} C_VEL
LIN {X 0,Y 88.861,Z 379.264,A -85,B 0,C 180,E1 -27846.387,E2 -27846.387} C_VEL
LIN {X 0,Y 94.555,Z 375.295,A -85,B 0,C 180,E1 -27851.99,E2 -27851.99} C_VEL
LIN {X 0,Y 101.033,Z 370.209,A -85,B 0,C 180,E1 -27856.924,E2 -27856.924} C_VEL
LIN {X 0,Y 108.303,Z 363.847,A -85,B 0,C 180,E1 -27861.146,E2 -27861.146} C_VEL
LIN {X 0,Y 116.175,Z 355.905,A -85,B 0,C 180,E1 -27864.758,E2 -27864.758} C_VEL
LIN {X 0,Y 123.009,Z 347.832,A -85,B 0,C 180,E1 -27867.434,E2 -27867.434} C_VEL
LIN {X 0,Y 130.18,Z 338.001,A -85,B 0,C 180,E1 -27869.749,E2 -27869.749} C_VEL
LIN {X 0,Y 136.826,Z 327.018,A -85,B 0,C 180,E1 -27871.601,E2 -27871.601} C_VEL
LIN {X 0,Y 142.084,Z 316.264,A -85,B 0,C 180,E1 -27872.921,E2 -27872.921} C_VEL
LIN {X 0,Y 146.238,Z 305.68,A -85,B 0,C 180,E1 -27873.874,E2 -27873.874} C_VEL
LIN {X 0,Y 150.057,Z 292.454,A -85,B 0,C 180,E1 -27874.772,E2 -27874.772} C_VEL
LIN {X 0,Y 152.444,Z 280.098,A -85,B 0,C 180,E1 -27875.305,E2 -27875.305} C_VEL
LIN {X 0,Y 153.262,Z 272.806,A -85,B 0,C 180,E1 -27875.567,E2 -27875.567} C_VEL
LIN {X 0,Y 150.872,Z 264.445,A -85,B 0,C 180,E1 -27879.067,E2 -27879.067} C_VEL
LIN {X 0,Y 148.863,Z 258.318,A -85,B 0,C 180,E1 -27882.551,E2 -27882.551} C_VEL
LIN {X 0,Y 146.946,Z 254.276,A -85,B 0,C 180,E1 -27886.517,E2 -27886.517} C_VEL
LIN {X 0,Y 146.663,Z 253.887,A -85,B 0,C 180,E1 -27887.182,E2 -27887.182} C_VEL
LIN {X 0,Y 145.775,Z 253.188,A -85,B 0,C 180,E1 -27889.453,E2 -27889.453} C_VEL
LIN {X 0,Y 144.968,Z 253.653,A -85,B 0,C 180,E1 -27891.772,E2 -27891.772} C_VEL
LIN {X 0,Y 143.801,Z 256.511,A -85,B 0,C 180,E1 -27898.062,E2 -27898.062} C_VEL
LIN {X 0,Y 143.847,Z 256.724,A -85,B 0,C 180,E1 -27899.668,E2 -27899.668} C_VEL
LIN {X 0,Y 144.403,Z 257.626,A -85,B 0,C 180,E1 -27903.624,E2 -27903.624} C_VEL
LIN {X 0,Y 146.02,Z 261.73,A -85,B 0,C 180,E1 -27909.174,E2 -27909.174} C_VEL
LIN {X 0,Y 147.857,Z 265.805,A -85,B 0,C 180,E1 -27913.049,E2 -27913.049} C_VEL
LIN {X 0,Y 150.158,Z 271.334,A -85,B 0,C 180,E1 -27916.847,E2 -27916.847} C_VEL
LIN {X 0,Y 150.639,Z 272.708,A -85,B 0,C 180,E1 -27917.599,E2 -27917.599} C_VEL
LIN {X 0,Y 148.328,Z 286.138,A -85,B 0,C 180,E1 -27918.237,E2 -27918.237} C_VEL
LIN {X 0,Y 144.982,Z 298.168,A -85,B 0,C 180,E1 -27919.028,E2 -27919.028} C_VEL
LIN {X 0,Y 140.393,Z 310.326,A -85,B 0,C 180,E1 -27920.177,E2 -27920.177} C_VEL
LIN {X 0,Y 135.114,Z 321.262,A -85,B 0,C 180,E1 -27921.595,E2 -27921.595} C_VEL
LIN {X 0,Y 129.145,Z 331.287,A -85,B 0,C 180,E1 -27923.312,E2 -27923.312} C_VEL
LIN {X 0,Y 122.592,Z 340.469,A -85,B 0,C 180,E1 -27925.45,E2 -27925.45} C_VEL
LIN {X 0,Y 115.478,Z 348.838,A -85,B 0,C 180,E1 -27928.053,E2 -27928.053} C_VEL
LIN {X 0,Y 107.35,Z 356.997,A -85,B 0,C 180,E1 -27931.665,E2 -27931.665} C_VEL
LIN {X 0,Y 99.761,Z 363.539,A -85,B 0,C 180,E1 -27935.884,E2 -27935.884} C_VEL
LIN {X 0,Y 92.601,Z 368.731,A -85,B 0,C 180,E1 -27940.622,E2 -27940.622} C_VEL
LIN {X 0,Y 86.18,Z 372.745,A -85,B 0,C 180,E1 -27946.112,E2 -27946.112} C_VEL
LIN {X 0,Y 80.59,Z 375.698,A -85,B 0,C 180,E1 -27952.373,E2 -27952.373} C_VEL
LIN {X 0,Y 77.448,Z 377.126,A -85,B 0,C 180,E1 -27957.007,E2 -27957.007} C_VEL
LIN {X 0,Y 72.676,Z 378.731,A -85,B 0,C 180,E1 -27967.239,E2 -27967.239} C_VEL
LIN {X 0,Y 71.21,Z 378.955,A -85,B 0,C 180,E1 -27972.772,E2 -27972.772} C_VEL
LIN {X 0,Y 70.329,Z 378.765,A -85,B 0,C 180,E1 -27978.466,E2 -27978.466} C_VEL
LIN {X 0,Y 69.979,Z 378.169,A -85,B 0,C 180,E1 -27984.231,E2 -27984.231} C_VEL
LIN {X 0,Y 70.369,Z 376.567,A -85,B 0,C 180,E1 -27992.86,E2 -27992.86} C_VEL
LIN {X 0,Y 72.837,Z 372.987,A -85,B 0,C 180,E1 -28003.953,E2 -28003.953} C_VEL
LIN {X 0,Y 76.046,Z 369.125,A -85,B 0,C 180,E1 -28011.69,E2 -28011.69} C_VEL
LIN {X 0,Y 80.401,Z 364.143,A -85,B 0,C 180,E1 -28018.73,E2 -28018.73} C_VEL
LIN {X 0,Y 85.754,Z 357.883,A -85,B 0,C 180,E1 -28025.002,E2 -28025.002} C_VEL
LIN {X 0,Y 91.956,Z 350.041,A -85,B 0,C 180,E1 -28030.508,E2 -28030.508} C_VEL
LIN {X 0,Y 97.632,Z 342.055,A -85,B 0,C 180,E1 -28034.569,E2 -28034.569} C_VEL
LIN {X 0,Y 103.688,Z 332.316,A -85,B 0,C 180,E1 -28038.203,E2 -28038.203} C_VEL
LIN {X 0,Y 109.427,Z 321.432,A -85,B 0,C 180,E1 -28041.138,E2 -28041.138} C_VEL
LIN {X 0,Y 114.048,Z 310.769,A -85,B 0,C 180,E1 -28043.229,E2 -28043.229} C_VEL
LIN {X 0,Y 118.404,Z 297.942,A -85,B 0,C 180,E1 -28045.063,E2 -28045.063} C_VEL
LIN {X 0,Y 121.603,Z 284.908,A -85,B 0,C 180,E1 -28046.341,E2 -28046.341} C_VEL
LIN {X 0,Y 123.67,Z 271.373,A -85,B 0,C 180,E1 -28047.166,E2 -28047.166} C_VEL
LIN {X 0,Y 125.551,Z 250.919,A -85,B 0,C 180,E1 -28048.028,E2 -28048.028} C_VEL
LIN {X 0,Y 122.581,Z 244.091,A -85,B 0,C 180,E1 -28051.522,E2 -28051.522} C_VEL
LIN {X 0,Y 119.39,Z 237.638,A -85,B 0,C 180,E1 -28055.954,E2 -28055.954} C_VEL
LIN {X 0,Y 117.437,Z 234.099,A -85,B 0,C 180,E1 -28059.242,E2 -28059.242} C_VEL
LIN {X 0,Y 115.68,Z 230.857,A -85,B 0,C 180,E1 -28062.946,E2 -28062.946} C_VEL
LIN {X 0,Y 113.882,Z 227.612,A -85,B 0,C 180,E1 -28068.348,E2 -28068.348} C_VEL
LIN {X 0,Y 113.697,Z 226.843,A -85,B 0,C 180,E1 -28069.313,E2 -28069.313} C_VEL
LIN {X 0,Y 112.754,Z 225.889,A -85,B 0,C 180,E1 -28076.426,E2 -28076.426} C_VEL
LIN {X 0,Y 112.99,Z 226.016,A -85,B 0,C 180,E1 -28081.113,E2 -28081.113} C_VEL
LIN {X 0,Y 113.784,Z 227.04,A -85,B 0,C 180,E1 -28085.482,E2 -28085.482} C_VEL
LIN {X 0,Y 115.517,Z 230.648,A -85,B 0,C 180,E1 -28091.071,E2 -28091.071} C_VEL
LIN {X 0,Y 116.209,Z 231.832,A -85,B 0,C 180,E1 -28092.664,E2 -28092.664} C_VEL
LIN {X 0,Y 118.329,Z 235.655,A -85,B 0,C 180,E1 -28096.719,E2 -28096.719} C_VEL
LIN {X 0,Y 121.113,Z 240.962,A -85,B 0,C 180,E1 -28100.93,E2 -28100.93} C_VEL
LIN {X 0,Y 122.497,Z 244.076,A -85,B 0,C 180,E1 -28102.784,E2 -28102.784} C_VEL
LIN {X 0,Y 124.949,Z 252.372,A -85,B 0,C 180,E1 -28106.033,E2 -28106.033} C_VEL
LIN {X 0,Y 125.349,Z 253.965,A -85,B 0,C 180,E1 -28106.549,E2 -28106.549} C_VEL
LIN {X 0,Y 122.498,Z 282.098,A -85,B 0,C 180,E1 -28107.694,E2 -28107.694} C_VEL
LIN {X 0,Y 119.989,Z 294.933,A -85,B 0,C 180,E1 -28108.537,E2 -28108.537} C_VEL
LIN {X 0,Y 116.435,Z 307.496,A -85,B 0,C 180,E1 -28109.818,E2 -28109.818} C_VEL
LIN {X 0,Y 112.172,Z 318.656,A -85,B 0,C 180,E1 -28111.396,E2 -28111.396} C_VEL
LIN {X 0,Y 106.636,Z 330.269,A -85,B 0,C 180,E1 -28113.695,E2 -28113.695} C_VEL
LIN {X 0,Y 100.76,Z 340.742,A -85,B 0,C 180,E1 -28116.674,E2 -28116.674} C_VEL
LIN {X 0,Y 94.506,Z 350.141,A -85,B 0,C 180,E1 -28120.344,E2 -28120.344} C_VEL
LIN {X 0,Y 87.748,Z 359.245,A -85,B 0,C 180,E1 -28125.515,E2 -28125.515} C_VEL
LIN {X 0,Y 82.683,Z 365.53,A -85,B 0,C 180,E1 -28130.509,E2 -28130.509} C_VEL
LIN {X 0,Y 77.653,Z 371.545,A -85,B 0,C 180,E1 -28137.116,E2 -28137.116} C_VEL
LIN {X 0,Y 73.657,Z 376.363,A -85,B 0,C 180,E1 -28144.579,E2 -28144.579} C_VEL
LIN {X 0,Y 71.097,Z 380.06,A -85,B 0,C 180,E1 -28152.755,E2 -28152.755} C_VEL
LIN {X 0,Y 70.143,Z 381.971,A -85,B 0,C 180,E1 -28158.446,E2 -28158.446} C_VEL
LIN {X 0,Y 69.794,Z 383.414,A -85,B 0,C 180,E1 -28164.226,E2 -28164.226} C_VEL
LIN {X 0,Y 69.954,Z 384.434,A -85,B 0,C 180,E1 -28170.005,E2 -28170.005} C_VEL
LIN {X 0,Y 69.796,Z 385.017,A -85,B 0,C 180,E1 -28175.784,E2 -28175.784} C_VEL
LIN {X 0,Y 70.172,Z 385.212,A -85,B 0,C 180,E1 -28181.56,E2 -28181.56} C_VEL
LIN {X 0,Y 71.166,Z 384.984,A -85,B 0,C 180,E1 -28187.239,E2 -28187.239} C_VEL
LIN {X 0,Y 75.026,Z 383.345,A -85,B 0,C 180,E1 -28197.934,E2 -28197.934} C_VEL
LIN {X 0,Y 77.954,Z 381.951,A -85,B 0,C 180,E1 -28202.752,E2 -28202.752} C_VEL
LIN {X 0,Y 83.236,Z 379.029,A -85,B 0,C 180,E1 -28209.296,E2 -28209.296} C_VEL
LIN {X 0,Y 89.377,Z 375.09,A -85,B 0,C 180,E1 -28215.053,E2 -28215.053} C_VEL
LIN {X 0,Y 96.312,Z 370.038,A -85,B 0,C 180,E1 -28220.019,E2 -28220.019} C_VEL
LIN {X 0,Y 103.997,Z 363.721,A -85,B 0,C 180,E1 -28224.193,E2 -28224.193} C_VEL
LIN {X 0,Y 112.214,Z 355.832,A -85,B 0,C 180,E1 -28227.731,E2 -28227.731} C_VEL
LIN {X 0,Y 119.336,Z 347.81,A -85,B 0,C 180,E1 -28230.309,E2 -28230.309} C_VEL
LIN {X 0,Y 126.756,Z 338.039,A -85,B 0,C 180,E1 -28232.519,E2 -28232.519} C_VEL
LIN {X 0,Y 133.6,Z 327.169,A -85,B 0,C 180,E1 -28234.275,E2 -28234.275} C_VEL
LIN {X 0,Y 139.006,Z 316.538,A -85,B 0,C 180,E1 -28235.518,E2 -28235.518} C_VEL
LIN {X 0,Y 143.563,Z 305.251,A -85,B 0,C 180,E1 -28236.479,E2 -28236.479} C_VEL
LIN {X 0,Y 147.541,Z 291.733,A -85,B 0,C 180,E1 -28237.347,E2 -28237.347} C_VEL
LIN {X 0,Y 150.004,Z 278.928,A -85,B 0,C 180,E1 -28237.848,E2 -28237.848} C_VEL
LIN {X 0,Y 150.35,Z 275.883,A -85,B 0,C 180,E1 -28237.981,E2 -28237.981} C_VEL
LIN {X 0,Y 148.586,Z 269.03,A -85,B 0,C 180,E1 -28241.087,E2 -28241.087} C_VEL
LIN {X 0,Y 147.119,Z 264.092,A -85,B 0,C 180,E1 -28244.057,E2 -28244.057} C_VEL
LIN {X 0,Y 145.527,Z 260.725,A -85,B 0,C 180,E1 -28247.785,E2 -28247.785} C_VEL
LIN {X 0,Y 144.219,Z 257.307,A -85,B 0,C 180,E1 -28253.003,E2 -28253.003} C_VEL
LIN {X 0,Y 143.847,Z 256.724,A -85,B 0,C 180,E1 -28259.668,E2 -28259.668} C_VEL
LIN {X 0,Y 143.979,Z 257.136,A -85,B 0,C 180,E1 -28261.217,E2 -28261.217} C_VEL
LIN {X 0,Y 144.205,Z 259.031,A -85,B 0,C 180,E1 -28263.441,E2 -28263.441} C_VEL
LIN {X 0,Y 144.479,Z 261.902,A -85,B 0,C 180,E1 -28265.512,E2 -28265.512} C_VEL
LIN {X 0,Y 145.826,Z 270.911,A -85,B 0,C 180,E1 -28270.923,E2 -28270.923} C_VEL
LIN {X 0,Y 147.548,Z 275.601,A -85,B 0,C 180,E1 -28274.516,E2 -28274.516} C_VEL
LIN {X 0,Y 147.861,Z 276.63,A -85,B 0,C 180,E1 -28275.176,E2 -28275.176} C_VEL
LIN {X 0,Y 145.013,Z 290.19,A -85,B 0,C 180,E1 -28275.839,E2 -28275.839} C_VEL
LIN {X 0,Y 140.99,Z 302.947,A -85,B 0,C 180,E1 -28276.747,E2 -28276.747} C_VEL
LIN {X 0,Y 135.956,Z 314.651,A -85,B 0,C 180,E1 -28277.888,E2 -28277.888} C_VEL
LIN {X 0,Y 130.275,Z 325.24,A -85,B 0,C 180,E1 -28279.359,E2 -28279.359} C_VEL
LIN {X 0,Y 123.442,Z 335.541,A -85,B 0,C 180,E1 -28281.2,E2 -28281.2} C_VEL
LIN {X 0,Y 116.707,Z 344.045,A -85,B 0,C 180,E1 -28283.309,E2 -28283.309} C_VEL
LIN {X 0,Y 109.396,Z 351.861,A -85,B 0,C 180,E1 -28285.913,E2 -28285.913} C_VEL
LIN {X 0,Y 101.031,Z 359.465,A -85,B 0,C 180,E1 -28289.59,E2 -28289.59} C_VEL
LIN {X 0,Y 93.11,Z 365.555,A -85,B 0,C 180,E1 -28293.866,E2 -28293.866} C_VEL
LIN {X 0,Y 85.705,Z 370.368,A -85,B 0,C 180,E1 -28298.823,E2 -28298.823} C_VEL
LIN {X 0,Y 79.025,Z 374.051,A -85,B 0,C 180,E1 -28304.64,E2 -28304.64} C_VEL
LIN {X 0,Y 75.034,Z 375.944,A -85,B 0,C 180,E1 -28309.025,E2 -28309.025} C_VEL
LIN {X 0,Y 71.539,Z 377.402,A -85,B 0,C 180,E1 -28313.877,E2 -28313.877} C_VEL
LIN {X 0,Y 66.127,Z 379.036,A -85,B 0,C 180,E1 -28324.836,E2 -28324.836} C_VEL
LIN {X 0,Y 64.421,Z 379.273,A -85,B 0,C 180,E1 -28330.89,E2 -28330.89} C_VEL
LIN {X 0,Y 63.343,Z 379.112,A -85,B 0,C 180,E1 -28337.173,E2 -28337.173} C_VEL
LIN {X 0,Y 62.904,Z 378.53,A -85,B 0,C 180,E1 -28343.579,E2 -28343.579} C_VEL
LIN {X 0,Y 63.481,Z 376.572,A -85,B 0,C 180,E1 -28354.856,E2 -28354.856} C_VEL
LIN {X 0,Y 65.975,Z 373.406,A -85,B 0,C 180,E1 -28365.439,E2 -28365.439} C_VEL
LIN {X 0,Y 69.529,Z 369.575,A -85,B 0,C 180,E1 -28373.842,E2 -28373.842} C_VEL
LIN {X 0,Y 74.274,Z 364.628,A -85,B 0,C 180,E1 -28381.354,E2 -28381.354} C_VEL
LIN {X 0,Y 80.061,Z 358.413,A -85,B 0,C 180,E1 -28387.907,E2 -28387.907} C_VEL
LIN {X 0,Y 86.707,Z 350.629,A -85,B 0,C 180,E1 -28393.542,E2 -28393.542} C_VEL
LIN {X 0,Y 93.99,Z 340.926,A -85,B 0,C 180,E1 -28398.388,E2 -28398.388} C_VEL
LIN {X 0,Y 100.471,Z 330.84,A -85,B 0,C 180,E1 -28401.894,E2 -28401.894} C_VEL
LIN {X 0,Y 106.476,Z 319.439,A -85,B 0,C 180,E1 -28404.761,E2 -28404.761} C_VEL
LIN {X 0,Y 111.35,Z 308.22,A -85,B 0,C 180,E1 -28406.743,E2 -28406.743} C_VEL
LIN {X 0,Y 115.228,Z 296.802,A -85,B 0,C 180,E1 -28408.213,E2 -28408.213} C_VEL
LIN {X 0,Y 118.443,Z 283.377,A -85,B 0,C 180,E1 -28409.432,E2 -28409.432} C_VEL
LIN {X 0,Y 120.387,Z 270.503,A -85,B 0,C 180,E1 -28410.139,E2 -28410.139} C_VEL
LIN {X 0,Y 121.949,Z 253.96,A -85,B 0,C 180,E1 -28410.832,E2 -28410.832} C_VEL
LIN {X 0,Y 118.9,Z 246.906,A -85,B 0,C 180,E1 -28415.063,E2 -28415.063} C_VEL
LIN {X 0,Y 116.727,Z 242.357,A -85,B 0,C 180,E1 -28418.708,E2 -28418.708} C_VEL
LIN {X 0,Y 115.166,Z 239.326,A -85,B 0,C 180,E1 -28421.886,E2 -28421.886} C_VEL
LIN {X 0,Y 114.314,Z 237.552,A -85,B 0,C 180,E1 -28424.008,E2 -28424.008} C_VEL
LIN {X 0,Y 112.667,Z 233.962,A -85,B 0,C 180,E1 -28429.871,E2 -28429.871} C_VEL
LIN {X 0,Y 111.969,Z 233.127,A -85,B 0,C 180,E1 -28434.597,E2 -28434.597} C_VEL
LIN {X 0,Y 112.062,Z 232.989,A -85,B 0,C 180,E1 -28440.561,E2 -28440.561} C_VEL
LIN {X 0,Y 112.71,Z 233.955,A -85,B 0,C 180,E1 -28444.694,E2 -28444.694} C_VEL
LIN {X 0,Y 114.732,Z 238.347,A -85,B 0,C 180,E1 -28451.449,E2 -28451.449} C_VEL
LIN {X 0,Y 116.696,Z 242.223,A -85,B 0,C 180,E1 -28455.612,E2 -28455.612} C_VEL
LIN {X 0,Y 119.165,Z 247.372,A -85,B 0,C 180,E1 -28459.711,E2 -28459.711} C_VEL
LIN {X 0,Y 120.171,Z 250.132,A -85,B 0,C 180,E1 -28461.243,E2 -28461.243} C_VEL
LIN {X 0,Y 121.787,Z 256.327,A -85,B 0,C 180,E1 -28463.712,E2 -28463.712} C_VEL
LIN {X 0,Y 119.107,Z 281.753,A -85,B 0,C 180,E1 -28464.743,E2 -28464.743} C_VEL
LIN {X 0,Y 116.375,Z 295.1,A -85,B 0,C 180,E1 -28465.575,E2 -28465.575} C_VEL
LIN {X 0,Y 112.687,Z 307.509,A -85,B 0,C 180,E1 -28466.803,E2 -28466.803} C_VEL
LIN {X 0,Y 107.903,Z 319.384,A -85,B 0,C 180,E1 -28468.452,E2 -28468.452} C_VEL
LIN {X 0,Y 102.145,Z 330.805,A -85,B 0,C 180,E1 -28470.686,E2 -28470.686} C_VEL
LIN {X 0,Y 95.996,Z 341.116,A -85,B 0,C 180,E1 -28473.623,E2 -28473.623} C_VEL
LIN {X 0,Y 88.775,Z 351.179,A -85,B 0,C 180,E1 -28477.667,E2 -28477.667} C_VEL
LIN {X 0,Y 81.664,Z 360.057,A -85,B 0,C 180,E1 -28482.994,E2 -28482.994} C_VEL
LIN {X 0,Y 76.537,Z 365.879,A -85,B 0,C 180,E1 -28487.975,E2 -28487.975} C_VEL
LIN {X 0,Y 71.744,Z 371.064,A -85,B 0,C 180,E1 -28494.009,E2 -28494.009} C_VEL
LIN {X 0,Y 67.295,Z 375.917,A -85,B 0,C 180,E1 -28501.975,E2 -28501.975} C_VEL
LIN {X 0,Y 64.292,Z 379.643,A -85,B 0,C 180,E1 -28510.863,E2 -28510.863} C_VEL
LIN {X 0,Y 63.166,Z 381.57,A -85,B 0,C 180,E1 -28517.149,E2 -28517.149} C_VEL
LIN {X 0,Y 62.713,Z 383.042,A -85,B 0,C 180,E1 -28523.572,E2 -28523.572} C_VEL
LIN {X 0,Y 62.85,Z 384.076,A -85,B 0,C 180,E1 -28530.006,E2 -28530.006} C_VEL
LIN {X 0,Y 62.735,Z 384.673,A -85,B 0,C 180,E1 -28536.438,E2 -28536.438} C_VEL
LIN {X 0,Y 63.196,Z 384.88,A -85,B 0,C 180,E1 -28542.857,E2 -28542.857} C_VEL
LIN {X 0,Y 64.4,Z 384.679,A -85,B 0,C 180,E1 -28549.116,E2 -28549.116} C_VEL
LIN {X 0,Y 68.816,Z 383.068,A -85,B 0,C 180,E1 -28560.712,E2 -28560.712} C_VEL
LIN {X 0,Y 72.068,Z 381.687,A -85,B 0,C 180,E1 -28565.816,E2 -28565.816} C_VEL
LIN {X 0,Y 77.856,Z 378.795,A -85,B 0,C 180,E1 -28572.617,E2 -28572.617} C_VEL
LIN {X 0,Y 84.48,Z 374.885,A -85,B 0,C 180,E1 -28578.486,E2 -28578.486} C_VEL
LIN {X 0,Y 91.895,Z 369.866,A -85,B 0,C 180,E1 -28583.426,E2 -28583.426} C_VEL
LIN {X 0,Y 100.006,Z 363.589,A -85,B 0,C 180,E1 -28587.497,E2 -28587.497} C_VEL
LIN {X 0,Y 108.584,Z 355.761,A -85,B 0,C 180,E1 -28590.906,E2 -28590.906} C_VEL
LIN {X 0,Y 115.985,Z 347.791,A -85,B 0,C 180,E1 -28593.355,E2 -28593.355} C_VEL
LIN {X 0,Y 124.414,Z 337.012,A -85,B 0,C 180,E1 -28595.633,E2 -28595.633} C_VEL
LIN {X 0,Y 131.452,Z 325.919,A -85,B 0,C 180,E1 -28597.264,E2 -28597.264} C_VEL
LIN {X 0,Y 136.226,Z 316.82,A -85,B 0,C 180,E1 -28598.227,E2 -28598.227} C_VEL
LIN {X 0,Y 140.796,Z 305.974,A -85,B 0,C 180,E1 -28599.098,E2 -28599.098} C_VEL
LIN {X 0,Y 144.69,Z 293.516,A -85,B 0,C 180,E1 -28599.871,E2 -28599.871} C_VEL
LIN {X 0,Y 147.566,Z 279.972,A -85,B 0,C 180,E1 -28600.396,E2 -28600.396} C_VEL
LIN {X 0,Y 147.61,Z 278.833,A -85,B 0,C 180,E1 -28600.585,E2 -28600.585} C_VEL
LIN {X 0,Y 146.402,Z 273.309,A -85,B 0,C 180,E1 -28603.359,E2 -28603.359} C_VEL
LIN {X 0,Y 145.553,Z 270.25,A -85,B 0,C 180,E1 -28605.38,E2 -28605.38} C_VEL
LIN {X 0,Y 144.356,Z 267.471,A -85,B 0,C 180,E1 -28608.548,E2 -28608.548} C_VEL
LIN {X 0,Y 143.26,Z 264.293,A -85,B 0,C 180,E1 -28613.486,E2 -28613.486} C_VEL
LIN {X 0,Y 143.011,Z 263.761,A -85,B 0,C 180,E1 -28620,E2 -28620} C_VEL
LIN {X 0,Y 143.416,Z 264.657,A -85,B 0,C 180,E1 -28623.134,E2 -28623.134} C_VEL
LIN {X 0,Y 144.79,Z 268.414,A -85,B 0,C 180,E1 -28628.373,E2 -28628.373} C_VEL
LIN {X 0,Y 145.826,Z 270.911,A -85,B 0,C 180,E1 -28630.923,E2 -28630.923} C_VEL
LIN {X 0,Y 146.085,Z 273.05,A -85,B 0,C 180,E1 -28631.855,E2 -28631.855} C_VEL
LIN {X 0,Y 145.971,Z 276.552,A -85,B 0,C 180,E1 -28632.562,E2 -28632.562} C_VEL
LIN {X 0,Y 145.533,Z 279.773,A -85,B 0,C 180,E1 -28632.868,E2 -28632.868} C_VEL
LIN {X 0,Y 142.761,Z 291.205,A -85,B 0,C 180,E1 -28633.184,E2 -28633.184} C_VEL
LIN {X 0,Y 139.199,Z 302.261,A -85,B 0,C 180,E1 -28633.923,E2 -28633.923} C_VEL
LIN {X 0,Y 134.517,Z 313.254,A -85,B 0,C 180,E1 -28634.858,E2 -28634.858} C_VEL
LIN {X 0,Y 128.983,Z 323.621,A -85,B 0,C 180,E1 -28636.113,E2 -28636.113} C_VEL
LIN {X 0,Y 121.814,Z 334.414,A -85,B 0,C 180,E1 -28637.825,E2 -28637.825} C_VEL
LIN {X 0,Y 114.072,Z 344.054,A -85,B 0,C 180,E1 -28640.015,E2 -28640.015} C_VEL
LIN {X 0,Y 106.467,Z 351.93,A -85,B 0,C 180,E1 -28642.452,E2 -28642.452} C_VEL
LIN {X 0,Y 97.374,Z 359.838,A -85,B 0,C 180,E1 -28646.067,E2 -28646.067} C_VEL
LIN {X 0,Y 89.321,Z 365.721,A -85,B 0,C 180,E1 -28650.052,E2 -28650.052} C_VEL
LIN {X 0,Y 81.402,Z 370.568,A -85,B 0,C 180,E1 -28654.889,E2 -28654.889} C_VEL
LIN {X 0,Y 74.175,Z 374.283,A -85,B 0,C 180,E1 -28660.706,E2 -28660.706} C_VEL
LIN {X 0,Y 69.779,Z 376.191,A -85,B 0,C 180,E1 -28665.162,E2 -28665.162} C_VEL
LIN {X 0,Y 65.88,Z 377.674,A -85,B 0,C 180,E1 -28670.196,E2 -28670.196} C_VEL
LIN {X 0,Y 59.723,Z 379.341,A -85,B 0,C 180,E1 -28681.914,E2 -28681.914} C_VEL
LIN {X 0,Y 57.71,Z 379.592,A -85,B 0,C 180,E1 -28688.565,E2 -28688.565} C_VEL
LIN {X 0,Y 56.413,Z 379.455,A -85,B 0,C 180,E1 -28695.566,E2 -28695.566} C_VEL
LIN {X 0,Y 55.827,Z 378.891,A -85,B 0,C 180,E1 -28702.761,E2 -28702.761} C_VEL
LIN {X 0,Y 56.578,Z 376.765,A -85,B 0,C 180,E1 -28716.404,E2 -28716.404} C_VEL
LIN {X 0,Y 58.643,Z 374.341,A -85,B 0,C 180,E1 -28725.683,E2 -28725.683} C_VEL
LIN {X 0,Y 63.113,Z 370.025,A -85,B 0,C 180,E1 -28736.443,E2 -28736.443} C_VEL
LIN {X 0,Y 68.344,Z 365.111,A -85,B 0,C 180,E1 -28744.435,E2 -28744.435} C_VEL
LIN {X 0,Y 74.613,Z 358.934,A -85,B 0,C 180,E1 -28751.243,E2 -28751.243} C_VEL
LIN {X 0,Y 81.727,Z 351.215,A -85,B 0,C 180,E1 -28756.958,E2 -28756.958} C_VEL
LIN {X 0,Y 89.455,Z 341.563,A -85,B 0,C 180,E1 -28761.772,E2 -28761.772} C_VEL
LIN {X 0,Y 96.272,Z 331.573,A -85,B 0,C 180,E1 -28765.204,E2 -28765.204} C_VEL
LIN {X 0,Y 102.567,Z 320.262,A -85,B 0,C 180,E1 -28767.981,E2 -28767.981} C_VEL
LIN {X 0,Y 107.644,Z 309.162,A -85,B 0,C 180,E1 -28769.884,E2 -28769.884} C_VEL
LIN {X 0,Y 112.046,Z 296.759,A -85,B 0,C 180,E1 -28771.411,E2 -28771.411} C_VEL
LIN {X 0,Y 115.377,Z 283.231,A -85,B 0,C 180,E1 -28772.571,E2 -28772.571} C_VEL
LIN {X 0,Y 117.316,Z 270.704,A -85,B 0,C 180,E1 -28773.22,E2 -28773.22} C_VEL
LIN {X 0,Y 118.618,Z 257.379,A -85,B 0,C 180,E1 -28773.78,E2 -28773.78} C_VEL
LIN {X 0,Y 116.14,Z 251.185,A -85,B 0,C 180,E1 -28777.9,E2 -28777.9} C_VEL
LIN {X 0,Y 114.067,Z 246.55,A -85,B 0,C 180,E1 -28782.217,E2 -28782.217} C_VEL
LIN {X 0,Y 112.952,Z 244.172,A -85,B 0,C 180,E1 -28785.203,E2 -28785.203} C_VEL
LIN {X 0,Y 111.584,Z 240.645,A -85,B 0,C 180,E1 -28790.979,E2 -28790.979} C_VEL
LIN {X 0,Y 111.022,Z 239.996,A -85,B 0,C 180,E1 -28796.37,E2 -28796.37} C_VEL
LIN {X 0,Y 111.222,Z 240.15,A -85,B 0,C 180,E1 -28800.905,E2 -28800.905} C_VEL
LIN {X 0,Y 111.69,Z 240.933,A -85,B 0,C 180,E1 -28804.059,E2 -28804.059} C_VEL
LIN {X 0,Y 113.443,Z 245.169,A -85,B 0,C 180,E1 -28810.579,E2 -28810.579} C_VEL
LIN {X 0,Y 115.107,Z 248.798,A -85,B 0,C 180,E1 -28814.474,E2 -28814.474} C_VEL
LIN {X 0,Y 117.331,Z 253.972,A -85,B 0,C 180,E1 -28818.555,E2 -28818.555} C_VEL
LIN {X 0,Y 118.552,Z 259.015,A -85,B 0,C 180,E1 -28820.779,E2 -28820.779} C_VEL
LIN {X 0,Y 115.999,Z 281.679,A -85,B 0,C 180,E1 -28821.642,E2 -28821.642} C_VEL
LIN {X 0,Y 113.096,Z 295.255,A -85,B 0,C 180,E1 -28822.438,E2 -28822.438} C_VEL
LIN {X 0,Y 109.273,Z 307.502,A -85,B 0,C 180,E1 -28823.59,E2 -28823.59} C_VEL
LIN {X 0,Y 103.942,Z 320.106,A -85,B 0,C 180,E1 -28825.275,E2 -28825.275} C_VEL
LIN {X 0,Y 97.975,Z 331.339,A -85,B 0,C 180,E1 -28827.425,E2 -28827.425} C_VEL
LIN {X 0,Y 91.531,Z 341.447,A -85,B 0,C 180,E1 -28830.263,E2 -28830.263} C_VEL
LIN {X 0,Y 84.605,Z 350.576,A -85,B 0,C 180,E1 -28833.84,E2 -28833.84} C_VEL
LIN {X 0,Y 76.973,Z 359.5,A -85,B 0,C 180,E1 -28839.104,E2 -28839.104} C_VEL
LIN {X 0,Y 71.954,Z 364.675,A -85,B 0,C 180,E1 -28843.385,E2 -28843.385} C_VEL
LIN {X 0,Y 68.091,Z 368.698,A -85,B 0,C 180,E1 -28847.872,E2 -28847.872} C_VEL
LIN {X 0,Y 62.611,Z 373.995,A -85,B 0,C 180,E1 -28855.866,E2 -28855.866} C_VEL
LIN {X 0,Y 58.557,Z 378.112,A -85,B 0,C 180,E1 -28865.168,E2 -28865.168} C_VEL
LIN {X 0,Y 56.241,Z 381.169,A -85,B 0,C 180,E1 -28875.534,E2 -28875.534} C_VEL
LIN {X 0,Y 55.629,Z 382.668,A -85,B 0,C 180,E1 -28882.749,E2 -28882.749} C_VEL
LIN {X 0,Y 55.753,Z 383.719,A -85,B 0,C 180,E1 -28890.007,E2 -28890.007} C_VEL
LIN {X 0,Y 55.658,Z 384.328,A -85,B 0,C 180,E1 -28897.261,E2 -28897.261} C_VEL
LIN {X 0,Y 56.276,Z 384.548,A -85,B 0,C 180,E1 -28904.47,E2 -28904.47} C_VEL
LIN {X 0,Y 57.692,Z 384.372,A -85,B 0,C 180,E1 -28911.442,E2 -28911.442} C_VEL
LIN {X 0,Y 62.803,Z 382.791,A -85,B 0,C 180,E1 -28924.03,E2 -28924.03} C_VEL
LIN {X 0,Y 66.415,Z 381.424,A -85,B 0,C 180,E1 -28929.42,E2 -28929.42} C_VEL
LIN {X 0,Y 72.775,Z 378.561,A -85,B 0,C 180,E1 -28936.416,E2 -28936.416} C_VEL
LIN {X 0,Y 79.935,Z 374.683,A -85,B 0,C 180,E1 -28942.313,E2 -28942.313} C_VEL
LIN {X 0,Y 87.844,Z 369.698,A -85,B 0,C 180,E1 -28947.152,E2 -28947.152} C_VEL
LIN {X 0,Y 96.365,Z 363.457,A -85,B 0,C 180,E1 -28951.071,E2 -28951.071} C_VEL
LIN {X 0,Y 105.309,Z 355.693,A -85,B 0,C 180,E1 -28954.289,E2 -28954.289} C_VEL
LIN {X 0,Y 112.983,Z 347.774,A -85,B 0,C 180,E1 -28956.57,E2 -28956.57} C_VEL
LIN {X 0,Y 121.659,Z 337.057,A -85,B 0,C 180,E1 -28958.678,E2 -28958.678} C_VEL
LIN {X 0,Y 128.877,Z 326.087,A -85,B 0,C 180,E1 -28960.174,E2 -28960.174} C_VEL
LIN {X 0,Y 133.764,Z 317.072,A -85,B 0,C 180,E1 -28961.043,E2 -28961.043} C_VEL
LIN {X 0,Y 138.986,Z 304.88,A -85,B 0,C 180,E1 -28961.934,E2 -28961.934} C_VEL
LIN {X 0,Y 143.099,Z 291.682,A -85,B 0,C 180,E1 -28962.658,E2 -28962.658} C_VEL
LIN {X 0,Y 145.116,Z 282.423,A -85,B 0,C 180,E1 -28963.008,E2 -28963.008} C_VEL
LIN {X 0,Y 144.286,Z 277.321,A -85,B 0,C 180,E1 -28965.904,E2 -28965.904} C_VEL
LIN {X 0,Y 143.203,Z 274.248,A -85,B 0,C 180,E1 -28969.265,E2 -28969.265} C_VEL
LIN {X 0,Y 142.325,Z 271.291,A -85,B 0,C 180,E1 -28973.888,E2 -28973.888} C_VEL
LIN {X 0,Y 142.141,Z 270.836,A -85,B 0,C 180,E1 -28980,E2 -28980} C_VEL
LIN {X 0,Y 142.449,Z 271.68,A -85,B 0,C 180,E1 -28982.696,E2 -28982.696} C_VEL
LIN {X 0,Y 143.491,Z 275.12,A -85,B 0,C 180,E1 -28987.564,E2 -28987.564} C_VEL
LIN {X 0,Y 144.604,Z 278.635,A -85,B 0,C 180,E1 -28991.033,E2 -28991.033} C_VEL
LIN {X 0,Y 145.209,Z 280.732,A -85,B 0,C 180,E1 -28992.67,E2 -28992.67} C_VEL
LIN {X 0,Y 142.761,Z 291.205,A -85,B 0,C 180,E1 -28993.184,E2 -28993.184} C_VEL
LIN {X 0,Y 140.916,Z 296.84,A -85,B 0,C 180,E1 -28993.225,E2 -28993.225} C_VEL
LIN {X 0,Y 136.921,Z 305.858,A -85,B 0,C 180,E1 -28992.683,E2 -28992.683} C_VEL
LIN {X 0,Y 132.274,Z 314.536,A -85,B 0,C 180,E1 -28992.268,E2 -28992.268} C_VEL
LIN {X 0,Y 129.388,Z 319.629,A -85,B 0,C 180,E1 -28992.549,E2 -28992.549} C_VEL
LIN {X 0,Y 122.274,Z 331.015,A -85,B 0,C 180,E1 -28994.077,E2 -28994.077} C_VEL
LIN {X 0,Y 115.024,Z 340.443,A -85,B 0,C 180,E1 -28995.769,E2 -28995.769} C_VEL
LIN {X 0,Y 107.077,Z 349.018,A -85,B 0,C 180,E1 -28997.871,E2 -28997.871} C_VEL
LIN {X 0,Y 97.79,Z 357.318,A -85,B 0,C 180,E1 -29000.879,E2 -29000.879} C_VEL
LIN {X 0,Y 88.886,Z 363.979,A -85,B 0,C 180,E1 -29004.587,E2 -29004.587} C_VEL
LIN {X 0,Y 80.289,Z 369.278,A -85,B 0,C 180,E1 -29008.907,E2 -29008.907} C_VEL
LIN {X 0,Y 72.248,Z 373.391,A -85,B 0,C 180,E1 -29014.216,E2 -29014.216} C_VEL
LIN {X 0,Y 64.886,Z 376.439,A -85,B 0,C 180,E1 -29020.687,E2 -29020.687} C_VEL
LIN {X 0,Y 60.544,Z 377.943,A -85,B 0,C 180,E1 -29025.847,E2 -29025.847} C_VEL
LIN {X 0,Y 56.731,Z 378.994,A -85,B 0,C 180,E1 -29031.719,E2 -29031.719} C_VEL
LIN {X 0,Y 51.107,Z 379.912,A -85,B 0,C 180,E1 -29045.627,E2 -29045.627} C_VEL
LIN {X 0,Y 49.527,Z 379.794,A -85,B 0,C 180,E1 -29053.505,E2 -29053.505} C_VEL
LIN {X 0,Y 48.787,Z 379.25,A -85,B 0,C 180,E1 -29061.71,E2 -29061.71} C_VEL
LIN {X 0,Y 48.797,Z 378.32,A -85,B 0,C 180,E1 -29069.992,E2 -29069.992} C_VEL
LIN {X 0,Y 49.826,Z 376.826,A -85,B 0,C 180,E1 -29079.112,E2 -29079.112} C_VEL
LIN {X 0,Y 53.746,Z 373.105,A -85,B 0,C 180,E1 -29093.089,E2 -29093.089} C_VEL
LIN {X 0,Y 59.301,Z 368.44,A -85,B 0,C 180,E1 -29103.583,E2 -29103.583} C_VEL
LIN {X 0,Y 65.307,Z 363.243,A -85,B 0,C 180,E1 -29111.122,E2 -29111.122} C_VEL
LIN {X 0,Y 73.204,Z 355.841,A -85,B 0,C 180,E1 -29118.068,E2 -29118.068} C_VEL
LIN {X 0,Y 81.1,Z 347.264,A -85,B 0,C 180,E1 -29123.274,E2 -29123.274} C_VEL
LIN {X 0,Y 88.11,Z 338.467,A -85,B 0,C 180,E1 -29126.871,E2 -29126.871} C_VEL
LIN {X 0,Y 95.325,Z 327.646,A -85,B 0,C 180,E1 -29130.021,E2 -29130.021} C_VEL
LIN {X 0,Y 101.272,Z 316.699,A -85,B 0,C 180,E1 -29132.219,E2 -29132.219} C_VEL
LIN {X 0,Y 106.568,Z 304.443,A -85,B 0,C 180,E1 -29133.958,E2 -29133.958} C_VEL
LIN {X 0,Y 110.596,Z 291.998,A -85,B 0,C 180,E1 -29135.221,E2 -29135.221} C_VEL
LIN {X 0,Y 113.339,Z 279.707,A -85,B 0,C 180,E1 -29136.041,E2 -29136.041} C_VEL
LIN {X 0,Y 115.639,Z 260.957,A -85,B 0,C 180,E1 -29136.835,E2 -29136.835} C_VEL
LIN {X 0,Y 113.707,Z 255.735,A -85,B 0,C 180,E1 -29140.76,E2 -29140.76} C_VEL
LIN {X 0,Y 112.289,Z 252.34,A -85,B 0,C 180,E1 -29144.357,E2 -29144.357} C_VEL
LIN {X 0,Y 111.567,Z 250.627,A -85,B 0,C 180,E1 -29146.686,E2 -29146.686} C_VEL
LIN {X 0,Y 110.517,Z 247.535,A -85,B 0,C 180,E1 -29152.106,E2 -29152.106} C_VEL
LIN {X 0,Y 110.156,Z 247.054,A -85,B 0,C 180,E1 -29156.342,E2 -29156.342} C_VEL
LIN {X 0,Y 110.402,Z 247.298,A -85,B 0,C 180,E1 -29161.367,E2 -29161.367} C_VEL
LIN {X 0,Y 110.65,Z 247.805,A -85,B 0,C 180,E1 -29163.186,E2 -29163.186} C_VEL
LIN {X 0,Y 112.04,Z 251.634,A -85,B 0,C 180,E1 -29169.25,E2 -29169.25} C_VEL
LIN {X 0,Y 113.518,Z 255.258,A -85,B 0,C 180,E1 -29173.196,E2 -29173.196} C_VEL
LIN {X 0,Y 115.203,Z 259.685,A -85,B 0,C 180,E1 -29176.73,E2 -29176.73} C_VEL
LIN {X 0,Y 115.58,Z 261.58,A -85,B 0,C 180,E1 -29177.585,E2 -29177.585} C_VEL
LIN {X 0,Y 113.229,Z 281.69,A -85,B 0,C 180,E1 -29178.377,E2 -29178.377} C_VEL
LIN {X 0,Y 110.247,Z 295.111,A -85,B 0,C 180,E1 -29179.1,E2 -29179.1} C_VEL
LIN {X 0,Y 106.49,Z 306.86,A -85,B 0,C 180,E1 -29180.14,E2 -29180.14} C_VEL
LIN {X 0,Y 101.113,Z 319.235,A -85,B 0,C 180,E1 -29181.632,E2 -29181.632} C_VEL
LIN {X 0,Y 94.896,Z 330.565,A -85,B 0,C 180,E1 -29183.593,E2 -29183.593} C_VEL
LIN {X 0,Y 88.152,Z 340.783,A -85,B 0,C 180,E1 -29186.255,E2 -29186.255} C_VEL
LIN {X 0,Y 80.838,Z 349.967,A -85,B 0,C 180,E1 -29189.622,E2 -29189.622} C_VEL
LIN {X 0,Y 72.674,Z 358.939,A -85,B 0,C 180,E1 -29194.725,E2 -29194.725} C_VEL
LIN {X 0,Y 65.217,Z 366.148,A -85,B 0,C 180,E1 -29201.042,E2 -29201.042} C_VEL
LIN {X 0,Y 58.741,Z 371.895,A -85,B 0,C 180,E1 -29208.858,E2 -29208.858} C_VEL
LIN {X 0,Y 53.491,Z 376.416,A -85,B 0,C 180,E1 -29218.304,E2 -29218.304} C_VEL
LIN {X 0,Y 51.004,Z 378.809,A -85,B 0,C 180,E1 -29225.591,E2 -29225.591} C_VEL
LIN {X 0,Y 49.35,Z 380.767,A -85,B 0,C 180,E1 -29233.46,E2 -29233.46} C_VEL
LIN {X 0,Y 48.579,Z 382.294,A -85,B 0,C 180,E1 -29241.69,E2 -29241.69} C_VEL
LIN {X 0,Y 48.646,Z 383.36,A -85,B 0,C 180,E1 -29250.008,E2 -29250.008} C_VEL
LIN {X 0,Y 48.604,Z 383.982,A -85,B 0,C 180,E1 -29258.322,E2 -29258.322} C_VEL
LIN {X 0,Y 49.421,Z 384.217,A -85,B 0,C 180,E1 -29266.531,E2 -29266.531} C_VEL
LIN {X 0,Y 51.107,Z 384.061,A -85,B 0,C 180,E1 -29274.373,E2 -29274.373} C_VEL
LIN {X 0,Y 57.048,Z 382.515,A -85,B 0,C 180,E1 -29288.031,E2 -29288.031} C_VEL
LIN {X 0,Y 65.61,Z 379.403,A -85,B 0,C 180,E1 -29298.583,E2 -29298.583} C_VEL
LIN {X 0,Y 73.227,Z 375.858,A -85,B 0,C 180,E1 -29304.841,E2 -29304.841} C_VEL
LIN {X 0,Y 81.316,Z 371.334,A -85,B 0,C 180,E1 -29309.808,E2 -29309.808} C_VEL
LIN {X 0,Y 91.616,Z 364.447,A -85,B 0,C 180,E1 -29314.345,E2 -29314.345} C_VEL
LIN {X 0,Y 100.864,Z 357.004,A -85,B 0,C 180,E1 -29317.411,E2 -29317.411} C_VEL
LIN {X 0,Y 108.752,Z 349.432,A -85,B 0,C 180,E1 -29319.569,E2 -29319.569} C_VEL
LIN {X 0,Y 116.844,Z 340.28,A -85,B 0,C 180,E1 -29321.33,E2 -29321.33} C_VEL
LIN {X 0,Y 124.206,Z 330.129,A -85,B 0,C 180,E1 -29322.723,E2 -29322.723} C_VEL
LIN {X 0,Y 129.995,Z 320.455,A -85,B 0,C 180,E1 -29323.672,E2 -29323.672} C_VEL
LIN {X 0,Y 134.626,Z 310.973,A -85,B 0,C 180,E1 -29324.426,E2 -29324.426} C_VEL
LIN {X 0,Y 139.214,Z 298.902,A -85,B 0,C 180,E1 -29325.119,E2 -29325.119} C_VEL
LIN {X 0,Y 142.75,Z 285.835,A -85,B 0,C 180,E1 -29325.65,E2 -29325.65} C_VEL
LIN {X 0,Y 142.417,Z 283.045,A -85,B 0,C 180,E1 -29327.532,E2 -29327.532} C_VEL
LIN {X 0,Y 141.768,Z 280.863,A -85,B 0,C 180,E1 -29330.214,E2 -29330.214} C_VEL
LIN {X 0,Y 141.238,Z 278.227,A -85,B 0,C 180,E1 -29334.401,E2 -29334.401} C_VEL
LIN {X 0,Y 141.107,Z 277.871,A -85,B 0,C 180,E1 -29340,E2 -29340} C_VEL
LIN {X 0,Y 141.268,Z 278.674,A -85,B 0,C 180,E1 -29342.317,E2 -29342.317} C_VEL
LIN {X 0,Y 141.968,Z 281.883,A -85,B 0,C 180,E1 -29346.931,E2 -29346.931} C_VEL
LIN {X 0,Y 142.635,Z 284.982,A -85,B 0,C 180,E1 -29350.039,E2 -29350.039} C_VEL
LIN {X 0,Y 139.655,Z 295.969,A -85,B 0,C 180,E1 -29350.645,E2 -29350.645} C_VEL
LIN {X 0,Y 135.339,Z 307.534,A -85,B 0,C 180,E1 -29351.422,E2 -29351.422} C_VEL
LIN {X 0,Y 129.388,Z 319.629,A -85,B 0,C 180,E1 -29352.549,E2 -29352.549} C_VEL
LIN {X 0,Y 126.283,Z 324.684,A -85,B 0,C 180,E1 -29352.883,E2 -29352.883} C_VEL
LIN {X 0,Y 120.315,Z 332.594,A -85,B 0,C 180,E1 -29352.676,E2 -29352.676} C_VEL
LIN {X 0,Y 113.802,Z 340.013,A -85,B 0,C 180,E1 -29352.53,E2 -29352.53} C_VEL
LIN {X 0,Y 109.848,Z 344.235,A -85,B 0,C 180,E1 -29353.037,E2 -29353.037} C_VEL
LIN {X 0,Y 101.867,Z 352.054,A -85,B 0,C 180,E1 -29354.997,E2 -29354.997} C_VEL
LIN {X 0,Y 92.094,Z 360.007,A -85,B 0,C 180,E1 -29357.96,E2 -29357.96} C_VEL
LIN {X 0,Y 83.086,Z 366.052,A -85,B 0,C 180,E1 -29361.484,E2 -29361.484} C_VEL
LIN {X 0,Y 74.158,Z 370.967,A -85,B 0,C 180,E1 -29365.791,E2 -29365.791} C_VEL
LIN {X 0,Y 65.731,Z 374.747,A -85,B 0,C 180,E1 -29371.19,E2 -29371.19} C_VEL
LIN {X 0,Y 60.462,Z 376.686,A -85,B 0,C 180,E1 -29375.535,E2 -29375.535} C_VEL
LIN {X 0,Y 55.624,Z 378.208,A -85,B 0,C 180,E1 -29380.695,E2 -29380.695} C_VEL
LIN {X 0,Y 51.302,Z 379.285,A -85,B 0,C 180,E1 -29386.758,E2 -29386.758} C_VEL
LIN {X 0,Y 44.685,Z 380.231,A -85,B 0,C 180,E1 -29401.838,E2 -29401.838} C_VEL
LIN {X 0,Y 42.737,Z 380.129,A -85,B 0,C 180,E1 -29410.789,E2 -29410.789} C_VEL
LIN {X 0,Y 41.737,Z 379.611,A -85,B 0,C 180,E1 -29420.297,E2 -29420.297} C_VEL
LIN {X 0,Y 41.701,Z 378.693,A -85,B 0,C 180,E1 -29429.991,E2 -29429.991} C_VEL
LIN {X 0,Y 43.552,Z 376.503,A -85,B 0,C 180,E1 -29444.476,E2 -29444.476} C_VEL
LIN {X 0,Y 48.995,Z 372.304,A -85,B 0,C 180,E1 -29460.127,E2 -29460.127} C_VEL
LIN {X 0,Y 54.955,Z 367.845,A -85,B 0,C 180,E1 -29469.74,E2 -29469.74} C_VEL
LIN {X 0,Y 63.362,Z 361.08,A -85,B 0,C 180,E1 -29478.468,E2 -29478.468} C_VEL
LIN {X 0,Y 71.42,Z 353.737,A -85,B 0,C 180,E1 -29484.265,E2 -29484.265} C_VEL
LIN {X 0,Y 80.008,Z 344.602,A -85,B 0,C 180,E1 -29488.91,E2 -29488.91} C_VEL
LIN {X 0,Y 88.208,Z 334.051,A -85,B 0,C 180,E1 -29492.412,E2 -29492.412} C_VEL
LIN {X 0,Y 95.086,Z 323.299,A -85,B 0,C 180,E1 -29494.87,E2 -29494.87} C_VEL
LIN {X 0,Y 100.532,Z 312.797,A -85,B 0,C 180,E1 -29496.558,E2 -29496.558} C_VEL
LIN {X 0,Y 105.643,Z 300.167,A -85,B 0,C 180,E1 -29497.992,E2 -29497.992} C_VEL
LIN {X 0,Y 109.406,Z 287.323,A -85,B 0,C 180,E1 -29499.057,E2 -29499.057} C_VEL
LIN {X 0,Y 111.906,Z 273.992,A -85,B 0,C 180,E1 -29499.713,E2 -29499.713} C_VEL
LIN {X 0,Y 112.937,Z 264.632,A -85,B 0,C 180,E1 -29500.133,E2 -29500.133} C_VEL
LIN {X 0,Y 111.491,Z 260.236,A -85,B 0,C 180,E1 -29503.917,E2 -29503.917} C_VEL
LIN {X 0,Y 110.433,Z 257.431,A -85,B 0,C 180,E1 -29507.513,E2 -29507.513} C_VEL
LIN {X 0,Y 109.571,Z 254.522,A -85,B 0,C 180,E1 -29512.629,E2 -29512.629} C_VEL
LIN {X 0,Y 109.289,Z 254.11,A -85,B 0,C 180,E1 -29516.313,E2 -29516.313} C_VEL
LIN {X 0,Y 109.484,Z 254.273,A -85,B 0,C 180,E1 -29520.919,E2 -29520.919} C_VEL
LIN {X 0,Y 109.697,Z 255.02,A -85,B 0,C 180,E1 -29522.869,E2 -29522.869} C_VEL
LIN {X 0,Y 110.783,Z 258.359,A -85,B 0,C 180,E1 -29528.206,E2 -29528.206} C_VEL
LIN {X 0,Y 111.99,Z 261.689,A -85,B 0,C 180,E1 -29531.883,E2 -29531.883} C_VEL
LIN {X 0,Y 112.97,Z 264.554,A -85,B 0,C 180,E1 -29534.294,E2 -29534.294} C_VEL
LIN {X 0,Y 111.201,Z 279.749,A -85,B 0,C 180,E1 -29534.9,E2 -29534.9} C_VEL
LIN {X 0,Y 108.309,Z 293.05,A -85,B 0,C 180,E1 -29535.494,E2 -29535.494} C_VEL
LIN {X 0,Y 104.076,Z 306.279,A -85,B 0,C 180,E1 -29536.512,E2 -29536.512} C_VEL
LIN {X 0,Y 98.717,Z 318.365,A -85,B 0,C 180,E1 -29537.8,E2 -29537.8} C_VEL
LIN {X 0,Y 92.283,Z 329.794,A -85,B 0,C 180,E1 -29539.548,E2 -29539.548} C_VEL
LIN {X 0,Y 85.215,Z 340.106,A -85,B 0,C 180,E1 -29541.914,E2 -29541.914} C_VEL
LIN {X 0,Y 77.562,Z 349.36,A -85,B 0,C 180,E1 -29545.04,E2 -29545.04} C_VEL
LIN {X 0,Y 68.845,Z 358.377,A -85,B 0,C 180,E1 -29549.818,E2 -29549.818} C_VEL
LIN {X 0,Y 60.722,Z 365.632,A -85,B 0,C 180,E1 -29555.897,E2 -29555.897} C_VEL
LIN {X 0,Y 53.561,Z 371.428,A -85,B 0,C 180,E1 -29563.817,E2 -29563.817} C_VEL
LIN {X 0,Y 47.56,Z 375.983,A -85,B 0,C 180,E1 -29573.777,E2 -29573.777} C_VEL
LIN {X 0,Y 44.604,Z 378.391,A -85,B 0,C 180,E1 -29581.801,E2 -29581.801} C_VEL
LIN {X 0,Y 42.558,Z 380.364,A -85,B 0,C 180,E1 -29590.724,E2 -29590.724} C_VEL
LIN {X 0,Y 41.541,Z 381.914,A -85,B 0,C 180,E1 -29600.269,E2 -29600.269} C_VEL
LIN {X 0,Y 41.539,Z 383.002,A -85,B 0,C 180,E1 -29610.009,E2 -29610.009} C_VEL
LIN {X 0,Y 41.589,Z 383.638,A -85,B 0,C 180,E1 -29619.738,E2 -29619.738} C_VEL
LIN {X 0,Y 44.703,Z 383.747,A -85,B 0,C 180,E1 -29638.15,E2 -29638.15} C_VEL
LIN {X 0,Y 47.72,Z 383.189,A -85,B 0,C 180,E1 -29646.102,E2 -29646.102} C_VEL
LIN {X 0,Y 56.118,Z 380.898,A -85,B 0,C 180,E1 -29658.722,E2 -29658.722} C_VEL
LIN {X 0,Y 63.772,Z 378.094,A -85,B 0,C 180,E1 -29665.754,E2 -29665.754} C_VEL
LIN {X 0,Y 72.102,Z 374.278,A -85,B 0,C 180,E1 -29671.322,E2 -29671.322} C_VEL
LIN {X 0,Y 81.008,Z 369.361,A -85,B 0,C 180,E1 -29675.645,E2 -29675.645} C_VEL
LIN {X 0,Y 90.347,Z 363.194,A -85,B 0,C 180,E1 -29678.991,E2 -29678.991} C_VEL
LIN {X 0,Y 99.961,Z 355.547,A -85,B 0,C 180,E1 -29681.66,E2 -29681.66} C_VEL
LIN {X 0,Y 109.793,Z 345.957,A -85,B 0,C 180,E1 -29683.783,E2 -29683.783} C_VEL
LIN {X 0,Y 118.09,Z 336.077,A -85,B 0,C 180,E1 -29685.272,E2 -29685.272} C_VEL
LIN {X 0,Y 125.636,Z 324.997,A -85,B 0,C 180,E1 -29686.406,E2 -29686.406} C_VEL
LIN {X 0,Y 130.565,Z 316.148,A -85,B 0,C 180,E1 -29687.088,E2 -29687.088} C_VEL
LIN {X 0,Y 136.134,Z 303.457,A -85,B 0,C 180,E1 -29687.771,E2 -29687.771} C_VEL
LIN {X 0,Y 140.276,Z 290.495,A -85,B 0,C 180,E1 -29688.289,E2 -29688.289} C_VEL
LIN {X 0,Y 140.49,Z 289.48,A -85,B 0,C 180,E1 -29688.457,E2 -29688.457} C_VEL
LIN {X 0,Y 140.06,Z 287.484,A -85,B 0,C 180,E1 -29690.979,E2 -29690.979} C_VEL
LIN {X 0,Y 139.756,Z 285.119,A -85,B 0,C 180,E1 -29694.879,E2 -29694.879} C_VEL
LIN {X 0,Y 139.665,Z 284.847,A -85,B 0,C 180,E1 -29700,E2 -29700} C_VEL
LIN {X 0,Y 139.718,Z 285.516,A -85,B 0,C 180,E1 -29701.802,E2 -29701.802} C_VEL
LIN {X 0,Y 140.055,Z 288.438,A -85,B 0,C 180,E1 -29706.122,E2 -29706.122} C_VEL
LIN {X 0,Y 140.208,Z 289.564,A -85,B 0,C 180,E1 -29707.434,E2 -29707.434} C_VEL
LIN {X 0,Y 136.306,Z 301.723,A -85,B 0,C 180,E1 -29708.101,E2 -29708.101} C_VEL
LIN {X 0,Y 131.584,Z 312.658,A -85,B 0,C 180,E1 -29708.836,E2 -29708.836} C_VEL
LIN {X 0,Y 125.905,Z 323.091,A -85,B 0,C 180,E1 -29709.818,E2 -29709.818} C_VEL
LIN {X 0,Y 119.07,Z 333.234,A -85,B 0,C 180,E1 -29711.093,E2 -29711.093} C_VEL
LIN {X 0,Y 111.645,Z 342.288,A -85,B 0,C 180,E1 -29712.642,E2 -29712.642} C_VEL
LIN {X 0,Y 109.848,Z 344.235,A -85,B 0,C 180,E1 -29713.037,E2 -29713.037} C_VEL
LIN {X 0,Y 105.709,Z 348.319,A -85,B 0,C 180,E1 -29713.632,E2 -29713.632} C_VEL
LIN {X 0,Y 98.079,Z 354.663,A -85,B 0,C 180,E1 -29713.81,E2 -29713.81} C_VEL
LIN {X 0,Y 90.025,Z 360.375,A -85,B 0,C 180,E1 -29714.161,E2 -29714.161} C_VEL
LIN {X 0,Y 85.253,Z 363.447,A -85,B 0,C 180,E1 -29715.185,E2 -29715.185} C_VEL
LIN {X 0,Y 74.428,Z 369.644,A -85,B 0,C 180,E1 -29719.206,E2 -29719.206} C_VEL
LIN {X 0,Y 65.272,Z 373.823,A -85,B 0,C 180,E1 -29723.752,E2 -29723.752} C_VEL
LIN {X 0,Y 55.931,Z 377.146,A -85,B 0,C 180,E1 -29730.175,E2 -29730.175} C_VEL
LIN {X 0,Y 46.348,Z 379.576,A -85,B 0,C 180,E1 -29740.685,E2 -29740.685} C_VEL
LIN {X 0,Y 38.533,Z 380.55,A -85,B 0,C 180,E1 -29756.816,E2 -29756.816} C_VEL
LIN {X 0,Y 36.057,Z 380.462,A -85,B 0,C 180,E1 -29767.045,E2 -29767.045} C_VEL
LIN {X 0,Y 34.737,Z 379.971,A -85,B 0,C 180,E1 -29778.317,E2 -29778.317} C_VEL
LIN {X 0,Y 34.594,Z 379.067,A -85,B 0,C 180,E1 -29789.989,E2 -29789.989} C_VEL
LIN {X 0,Y 37.288,Z 376.503,A -85,B 0,C 180,E1 -29809.537,E2 -29809.537} C_VEL
LIN {X 0,Y 43.011,Z 372.737,A -85,B 0,C 180,E1 -29824.871,E2 -29824.871} C_VEL
LIN {X 0,Y 49.719,Z 368.309,A -85,B 0,C 180,E1 -29834.961,E2 -29834.961} C_VEL
LIN {X 0,Y 58.912,Z 361.598,A -85,B 0,C 180,E1 -29843.622,E2 -29843.622} C_VEL
LIN {X 0,Y 67.535,Z 354.297,A -85,B 0,C 180,E1 -29849.14,E2 -29849.14} C_VEL
LIN {X 0,Y 76.601,Z 345.232,A -85,B 0,C 180,E1 -29853.438,E2 -29853.438} C_VEL
LIN {X 0,Y 85.169,Z 334.749,A -85,B 0,C 180,E1 -29856.624,E2 -29856.624} C_VEL
LIN {X 0,Y 92.315,Z 324.08,A -85,B 0,C 180,E1 -29858.831,E2 -29858.831} C_VEL
LIN {X 0,Y 97.941,Z 313.725,A -85,B 0,C 180,E1 -29860.346,E2 -29860.346} C_VEL
LIN {X 0,Y 103.211,Z 301.282,A -85,B 0,C 180,E1 -29861.618,E2 -29861.618} C_VEL
LIN {X 0,Y 107.228,Z 288.213,A -85,B 0,C 180,E1 -29862.609,E2 -29862.609} C_VEL
LIN {X 0,Y 109.722,Z 276.023,A -85,B 0,C 180,E1 -29863.167,E2 -29863.167} C_VEL
LIN {X 0,Y 110.627,Z 268.56,A -85,B 0,C 180,E1 -29863.512,E2 -29863.512} C_VEL
LIN {X 0,Y 109.601,Z 265.224,A -85,B 0,C 180,E1 -29867.092,E2 -29867.092} C_VEL
LIN {X 0,Y 108.641,Z 261.591,A -85,B 0,C 180,E1 -29873.033,E2 -29873.033} C_VEL
LIN {X 0,Y 108.423,Z 261.166,A -85,B 0,C 180,E1 -29876.283,E2 -29876.283} C_VEL
LIN {X 0,Y 108.613,Z 261.349,A -85,B 0,C 180,E1 -29880.926,E2 -29880.926} C_VEL
LIN {X 0,Y 109.541,Z 264.964,A -85,B 0,C 180,E1 -29887.025,E2 -29887.025} C_VEL
LIN {X 0,Y 110.629,Z 268.516,A -85,B 0,C 180,E1 -29890.871,E2 -29890.871} C_VEL
LIN {X 0,Y 110.459,Z 270.57,A -85,B 0,C 180,E1 -29891.061,E2 -29891.061} C_VEL
LIN {X 0,Y 108.32,Z 284.581,A -85,B 0,C 180,E1 -29891.487,E2 -29891.487} C_VEL
LIN {X 0,Y 105.099,Z 296.967,A -85,B 0,C 180,E1 -29892.086,E2 -29892.086} C_VEL
LIN {X 0,Y 100.936,Z 308.456,A -85,B 0,C 180,E1 -29892.91,E2 -29892.91} C_VEL
LIN {X 0,Y 95.113,Z 320.67,A -85,B 0,C 180,E1 -29894.131,E2 -29894.131} C_VEL
LIN {X 0,Y 88.501,Z 331.543,A -85,B 0,C 180,E1 -29895.681,E2 -29895.681} C_VEL
LIN {X 0,Y 81.207,Z 341.417,A -85,B 0,C 180,E1 -29897.844,E2 -29897.844} C_VEL
LIN {X 0,Y 73.248,Z 350.393,A -85,B 0,C 180,E1 -29900.708,E2 -29900.708} C_VEL
LIN {X 0,Y 64.098,Z 359.173,A -85,B 0,C 180,E1 -29905.251,E2 -29905.251} C_VEL
LIN {X 0,Y 55.457,Z 366.17,A -85,B 0,C 180,E1 -29911.208,E2 -29911.208} C_VEL
LIN {X 0,Y 46.459,Z 372.599,A -85,B 0,C 180,E1 -29920.869,E2 -29920.869} C_VEL
LIN {X 0,Y 40.103,Z 376.81,A -85,B 0,C 180,E1 -29932.179,E2 -29932.179} C_VEL
LIN {X 0,Y 35.911,Z 379.962,A -85,B 0,C 180,E1 -29946.969,E2 -29946.969} C_VEL
LIN {X 0,Y 34.535,Z 381.53,A -85,B 0,C 180,E1 -29958.269,E2 -29958.269} C_VEL
LIN {X 0,Y 34.425,Z 382.643,A -85,B 0,C 180,E1 -29970.011,E2 -29970.011} C_VEL
LIN {X 0,Y 34.597,Z 383.292,A -85,B 0,C 180,E1 -29981.731,E2 -29981.731} C_VEL
LIN {X 0,Y 38.565,Z 383.43,A -85,B 0,C 180,E1 -30003.152,E2 -30003.152} C_VEL
LIN {X 0,Y 42.163,Z 382.898,A -85,B 0,C 180,E1 -30011.827,E2 -30011.827} C_VEL
LIN {X 0,Y 51.689,Z 380.635,A -85,B 0,C 180,E1 -30024.678,E2 -30024.678} C_VEL
LIN {X 0,Y 60.037,Z 377.86,A -85,B 0,C 180,E1 -30031.408,E2 -30031.408} C_VEL
LIN {X 0,Y 68.964,Z 374.076,A -85,B 0,C 180,E1 -30036.527,E2 -30036.527} C_VEL
LIN {X 0,Y 78.348,Z 369.192,A -85,B 0,C 180,E1 -30040.381,E2 -30040.381} C_VEL
LIN {X 0,Y 88.051,Z 363.062,A -85,B 0,C 180,E1 -30043.309,E2 -30043.309} C_VEL
LIN {X 0,Y 97.956,Z 355.463,A -85,B 0,C 180,E1 -30045.61,E2 -30045.61} C_VEL
LIN {X 0,Y 106.337,Z 347.71,A -85,B 0,C 180,E1 -30047.135,E2 -30047.135} C_VEL
LIN {X 0,Y 115.64,Z 337.191,A -85,B 0,C 180,E1 -30048.531,E2 -30048.531} C_VEL
LIN {X 0,Y 123.298,Z 326.501,A -85,B 0,C 180,E1 -30049.511,E2 -30049.511} C_VEL
LIN {X 0,Y 129.098,Z 316.514,A -85,B 0,C 180,E1 -30050.139,E2 -30050.139} C_VEL
LIN {X 0,Y 134.388,Z 305.035,A -85,B 0,C 180,E1 -30050.662,E2 -30050.662} C_VEL
LIN {X 0,Y 137.646,Z 295.866,A -85,B 0,C 180,E1 -30051.028,E2 -30051.028} C_VEL
LIN {X 0,Y 138.086,Z 294.335,A -85,B 0,C 180,E1 -30051.218,E2 -30051.218} C_VEL
LIN {X 0,Y 137.918,Z 291.942,A -85,B 0,C 180,E1 -30055.25,E2 -30055.25} C_VEL
LIN {X 0,Y 137.847,Z 291.732,A -85,B 0,C 180,E1 -30060,E2 -30060} C_VEL
LIN {X 0,Y 137.79,Z 292.738,A -85,B 0,C 180,E1 -30062.01,E2 -30062.01} C_VEL
LIN {X 0,Y 137.839,Z 294.425,A -85,B 0,C 180,E1 -30064.754,E2 -30064.754} C_VEL
LIN {X 0,Y 132.831,Z 307.743,A -85,B 0,C 180,E1 -30065.452,E2 -30065.452} C_VEL
LIN {X 0,Y 127.257,Z 318.896,A -85,B 0,C 180,E1 -30066.217,E2 -30066.217} C_VEL
LIN {X 0,Y 120.458,Z 329.655,A -85,B 0,C 180,E1 -30067.303,E2 -30067.303} C_VEL
LIN {X 0,Y 113.665,Z 338.446,A -85,B 0,C 180,E1 -30068.377,E2 -30068.377} C_VEL
LIN {X 0,Y 105.262,Z 347.479,A -85,B 0,C 180,E1 -30069.985,E2 -30069.985} C_VEL
LIN {X 0,Y 95.29,Z 356.27,A -85,B 0,C 180,E1 -30072.234,E2 -30072.234} C_VEL
LIN {X 0,Y 85.253,Z 363.447,A -85,B 0,C 180,E1 -30075.185,E2 -30075.185} C_VEL
LIN {X 0,Y 80.361,Z 366.342,A -85,B 0,C 180,E1 -30076.373,E2 -30076.373} C_VEL
LIN {X 0,Y 71.514,Z 370.654,A -85,B 0,C 180,E1 -30077.348,E2 -30077.348} C_VEL
LIN {X 0,Y 62.392,Z 374.25,A -85,B 0,C 180,E1 -30078.633,E2 -30078.633} C_VEL
LIN {X 0,Y 57.16,Z 375.978,A -85,B 0,C 180,E1 -30080.649,E2 -30080.649} C_VEL
LIN {X 0,Y 47.543,Z 378.732,A -85,B 0,C 180,E1 -30087.493,E2 -30087.493} C_VEL
LIN {X 0,Y 42.038,Z 379.865,A -85,B 0,C 180,E1 -30093.274,E2 -30093.274} C_VEL
LIN {X 0,Y 32.792,Z 380.869,A -85,B 0,C 180,E1 -30109.972,E2 -30109.972} C_VEL
LIN {X 0,Y 29.613,Z 380.795,A -85,B 0,C 180,E1 -30121.649,E2 -30121.649} C_VEL
LIN {X 0,Y 27.792,Z 380.33,A -85,B 0,C 180,E1 -30135.338,E2 -30135.338} C_VEL
LIN {X 0,Y 27.486,Z 379.441,A -85,B 0,C 180,E1 -30149.987,E2 -30149.987} C_VEL
LIN {X 0,Y 28.78,Z 378.167,A -85,B 0,C 180,E1 -30164.121,E2 -30164.121} C_VEL
LIN {X 0,Y 33.186,Z 375.492,A -85,B 0,C 180,E1 -30181.954,E2 -30181.954} C_VEL
LIN {X 0,Y 39.815,Z 371.817,A -85,B 0,C 180,E1 -30194.902,E2 -30194.902} C_VEL
LIN {X 0,Y 47.768,Z 367.037,A -85,B 0,C 180,E1 -30204.003,E2 -30204.003} C_VEL
LIN {X 0,Y 56.512,Z 361.009,A -85,B 0,C 180,E1 -30210.506,E2 -30210.506} C_VEL
LIN {X 0,Y 65.765,Z 353.512,A -85,B 0,C 180,E1 -30215.264,E2 -30215.264} C_VEL
LIN {X 0,Y 73.708,Z 345.852,A -85,B 0,C 180,E1 -30218.364,E2 -30218.364} C_VEL
LIN {X 0,Y 82.623,Z 335.447,A -85,B 0,C 180,E1 -30221.122,E2 -30221.122} C_VEL
LIN {X 0,Y 90.011,Z 324.854,A -85,B 0,C 180,E1 -30223.016,E2 -30223.016} C_VEL
LIN {X 0,Y 95.8,Z 314.615,A -85,B 0,C 180,E1 -30224.319,E2 -30224.319} C_VEL
LIN {X 0,Y 101.213,Z 302.395,A -85,B 0,C 180,E1 -30225.4,E2 -30225.4} C_VEL
LIN {X 0,Y 105.518,Z 288.951,A -85,B 0,C 180,E1 -30226.299,E2 -30226.299} C_VEL
LIN {X 0,Y 108.266,Z 275.811,A -85,B 0,C 180,E1 -30226.816,E2 -30226.816} C_VEL
LIN {X 0,Y 108.63,Z 272.831,A -85,B 0,C 180,E1 -30227.044,E2 -30227.044} C_VEL
LIN {X 0,Y 108.053,Z 270.62,A -85,B 0,C 180,E1 -30230.169,E2 -30230.169} C_VEL
LIN {X 0,Y 107.647,Z 268.413,A -85,B 0,C 180,E1 -30234.38,E2 -30234.38} C_VEL
LIN {X 0,Y 107.699,Z 268.345,A -85,B 0,C 180,E1 -30240.467,E2 -30240.467} C_VEL
LIN {X 0,Y 108.342,Z 271.611,A -85,B 0,C 180,E1 -30245.817,E2 -30245.817} C_VEL
LIN {X 0,Y 108.701,Z 272.92,A -85,B 0,C 180,E1 -30247.482,E2 -30247.482} C_VEL
LIN {X 0,Y 106.414,Z 286.094,A -85,B 0,C 180,E1 -30247.87,E2 -30247.87} C_VEL
LIN {X 0,Y 102.937,Z 298.5,A -85,B 0,C 180,E1 -30248.366,E2 -30248.366} C_VEL
LIN {X 0,Y 98.731,Z 309.437,A -85,B 0,C 180,E1 -30249.037,E2 -30249.037} C_VEL
LIN {X 0,Y 92.782,Z 321.343,A -85,B 0,C 180,E1 -30250.058,E2 -30250.058} C_VEL
LIN {X 0,Y 85.166,Z 333.176,A -85,B 0,C 180,E1 -30251.523,E2 -30251.523} C_VEL
LIN {X 0,Y 77.654,Z 342.721,A -85,B 0,C 180,E1 -30253.389,E2 -30253.389} C_VEL
LIN {X 0,Y 69.411,Z 351.426,A -85,B 0,C 180,E1 -30255.889,E2 -30255.889} C_VEL
LIN {X 0,Y 59.815,Z 359.883,A -85,B 0,C 180,E1 -30259.976,E2 -30259.976} C_VEL
LIN {X 0,Y 52.091,Z 365.665,A -85,B 0,C 180,E1 -30264.418,E2 -30264.418} C_VEL
LIN {X 0,Y 44.857,Z 370.483,A -85,B 0,C 180,E1 -30270.508,E2 -30270.508} C_VEL
LIN {X 0,Y 37.021,Z 375.11,A -85,B 0,C 180,E1 -30280.61,E2 -30280.61} C_VEL
LIN {X 0,Y 30.93,Z 378.635,A -85,B 0,C 180,E1 -30295.401,E2 -30295.401} C_VEL
LIN {X 0,Y 27.608,Z 381.144,A -85,B 0,C 180,E1 -30315.266,E2 -30315.266} C_VEL
LIN {X 0,Y 27.331,Z 382.285,A -85,B 0,C 180,E1 -30330.014,E2 -30330.014} C_VEL
LIN {X 0,Y 27.661,Z 382.947,A -85,B 0,C 180,E1 -30344.733,E2 -30344.733} C_VEL
LIN {X 0,Y 32.835,Z 383.112,A -85,B 0,C 180,E1 -30369.963,E2 -30369.963} C_VEL
LIN {X 0,Y 37.15,Z 382.607,A -85,B 0,C 180,E1 -30379.189,E2 -30379.189} C_VEL
LIN {X 0,Y 47.918,Z 380.372,A -85,B 0,C 180,E1 -30391.657,E2 -30391.657} C_VEL
LIN {X 0,Y 56.962,Z 377.626,A -85,B 0,C 180,E1 -30397.737,E2 -30397.737} C_VEL
LIN {X 0,Y 66.447,Z 373.874,A -85,B 0,C 180,E1 -30402.176,E2 -30402.176} C_VEL
LIN {X 0,Y 76.25,Z 369.024,A -85,B 0,C 180,E1 -30405.434,E2 -30405.434} C_VEL
LIN {X 0,Y 86.281,Z 362.931,A -85,B 0,C 180,E1 -30407.828,E2 -30407.828} C_VEL
LIN {X 0,Y 96.438,Z 355.373,A -85,B 0,C 180,E1 -30409.698,E2 -30409.698} C_VEL
LIN {X 0,Y 104.987,Z 347.672,A -85,B 0,C 180,E1 -30410.907,E2 -30410.907} C_VEL
LIN {X 0,Y 113.58,Z 338.306,A -85,B 0,C 180,E1 -30411.922,E2 -30411.922} C_VEL
LIN {X 0,Y 121.348,Z 327.913,A -85,B 0,C 180,E1 -30412.681,E2 -30412.681} C_VEL
LIN {X 0,Y 127.409,Z 317.962,A -85,B 0,C 180,E1 -30413.184,E2 -30413.184} C_VEL
LIN {X 0,Y 133.422,Z 305.449,A -85,B 0,C 180,E1 -30413.666,E2 -30413.666} C_VEL
LIN {X 0,Y 135.18,Z 300.901,A -85,B 0,C 180,E1 -30413.826,E2 -30413.826} C_VEL
LIN {X 0,Y 135.65,Z 299.546,A -85,B 0,C 180,E1 -30414.053,E2 -30414.053} C_VEL
LIN {X 0,Y 135.651,Z 298.492,A -85,B 0,C 180,E1 -30417.031,E2 -30417.031} C_VEL
LIN {X 0,Y 135.657,Z 298.516,A -85,B 0,C 180,E1 -30420,E2 -30420} C_VEL
LIN {X 0,Y 135.469,Z 299.566,A -85,B 0,C 180,E1 -30421.86,E2 -30421.86} C_VEL
LIN {X 0,Y 134.508,Z 302.135,A -85,B 0,C 180,E1 -30422.132,E2 -30422.132} C_VEL
LIN {X 0,Y 129.51,Z 313.37,A -85,B 0,C 180,E1 -30422.675,E2 -30422.675} C_VEL
LIN {X 0,Y 123.161,Z 324.527,A -85,B 0,C 180,E1 -30423.45,E2 -30423.45} C_VEL
LIN {X 0,Y 115.435,Z 335.268,A -85,B 0,C 180,E1 -30424.445,E2 -30424.445} C_VEL
LIN {X 0,Y 105.974,Z 345.87,A -85,B 0,C 180,E1 -30425.835,E2 -30425.835} C_VEL
LIN {X 0,Y 95.73,Z 355.003,A -85,B 0,C 180,E1 -30427.628,E2 -30427.628} C_VEL
LIN {X 0,Y 85.614,Z 362.331,A -85,B 0,C 180,E1 -30429.89,E2 -30429.89} C_VEL
LIN {X 0,Y 75.674,Z 368.183,A -85,B 0,C 180,E1 -30432.78,E2 -30432.78} C_VEL
LIN {X 0,Y 65.917,Z 372.78,A -85,B 0,C 180,E1 -30436.332,E2 -30436.332} C_VEL
LIN {X 0,Y 57.16,Z 375.978,A -85,B 0,C 180,E1 -30440.649,E2 -30440.649} C_VEL
LIN {X 0,Y 51.937,Z 377.565,A -85,B 0,C 180,E1 -30443.102,E2 -30443.102} C_VEL
LIN {X 0,Y 42.604,Z 379.552,A -85,B 0,C 180,E1 -30446.418,E2 -30446.418} C_VEL
LIN {X 0,Y 33.397,Z 380.818,A -85,B 0,C 180,E1 -30451.659,E2 -30451.659} C_VEL
LIN {X 0,Y 28.683,Z 381.121,A -85,B 0,C 180,E1 -30458.204,E2 -30458.204} C_VEL
LIN {X 0,Y 23.584,Z 381.127,A -85,B 0,C 180,E1 -30473.397,E2 -30473.397} C_VEL
LIN {X 0,Y 20.967,Z 380.684,A -85,B 0,C 180,E1 -30490.397,E2 -30490.397} C_VEL
LIN {X 0,Y 20.371,Z 379.815,A -85,B 0,C 180,E1 -30509.982,E2 -30509.982} C_VEL
LIN {X 0,Y 21.98,Z 378.553,A -85,B 0,C 180,E1 -30528.63,E2 -30528.63} C_VEL
LIN {X 0,Y 27.668,Z 375.802,A -85,B 0,C 180,E1 -30550.353,E2 -30550.353} C_VEL
LIN {X 0,Y 35.159,Z 372.265,A -85,B 0,C 180,E1 -30563.07,E2 -30563.07} C_VEL
LIN {X 0,Y 43.984,Z 367.519,A -85,B 0,C 180,E1 -30571.48,E2 -30571.48} C_VEL
LIN {X 0,Y 55.004,Z 360.417,A -85,B 0,C 180,E1 -30577.853,E2 -30577.853} C_VEL
LIN {X 0,Y 64.779,Z 352.657,A -85,B 0,C 180,E1 -30581.658,E2 -30581.658} C_VEL
LIN {X 0,Y 74.752,Z 342.967,A -85,B 0,C 180,E1 -30584.489,E2 -30584.489} C_VEL
LIN {X 0,Y 83.146,Z 332.917,A -85,B 0,C 180,E1 -30586.399,E2 -30586.399} C_VEL
LIN {X 0,Y 90.731,Z 321.545,A -85,B 0,C 180,E1 -30587.917,E2 -30587.917} C_VEL
LIN {X 0,Y 96.689,Z 310.361,A -85,B 0,C 180,E1 -30588.87,E2 -30588.87} C_VEL
LIN {X 0,Y 101.462,Z 298.757,A -85,B 0,C 180,E1 -30589.61,E2 -30589.61} C_VEL
LIN {X 0,Y 105.188,Z 286.052,A -85,B 0,C 180,E1 -30590.244,E2 -30590.244} C_VEL
LIN {X 0,Y 106.919,Z 277.629,A -85,B 0,C 180,E1 -30590.581,E2 -30590.581} C_VEL
LIN {X 0,Y 106.669,Z 275.414,A -85,B 0,C 180,E1 -30594.802,E2 -30594.802} C_VEL
LIN {X 0,Y 106.712,Z 275.572,A -85,B 0,C 180,E1 -30600.235,E2 -30600.235} C_VEL
LIN {X 0,Y 106.989,Z 277.602,A -85,B 0,C 180,E1 -30603.845,E2 -30603.845} C_VEL
LIN {X 0,Y 104.139,Z 290.68,A -85,B 0,C 180,E1 -30604.185,E2 -30604.185} C_VEL
LIN {X 0,Y 100.223,Z 302.706,A -85,B 0,C 180,E1 -30604.693,E2 -30604.693} C_VEL
LIN {X 0,Y 95.273,Z 313.992,A -85,B 0,C 180,E1 -30605.272,E2 -30605.272} C_VEL
LIN {X 0,Y 89.212,Z 324.825,A -85,B 0,C 180,E1 -30606.015,E2 -30606.015} C_VEL
LIN {X 0,Y 81.456,Z 335.877,A -85,B 0,C 180,E1 -30607.194,E2 -30607.194} C_VEL
LIN {X 0,Y 72.899,Z 345.757,A -85,B 0,C 180,E1 -30608.859,E2 -30608.859} C_VEL
LIN {X 0,Y 64.429,Z 353.858,A -85,B 0,C 180,E1 -30611.001,E2 -30611.001} C_VEL
LIN {X 0,Y 54.127,Z 362.045,A -85,B 0,C 180,E1 -30614.716,E2 -30614.716} C_VEL
